TRANSITION not_3621:
NOT MP.ST03.SGM_3621
END_TRANSITION

TRANSITION StateOk:
(*ST08_408_Y54_4.State=STATE_OK*)

ST08_400_Y52_5.State=STATE_OK AND
gTipImp
END_TRANSITION

TRANSITION StateOk:
ST08_408_Y54_4.State =STATE_OK AND
gTipImp
END_TRANSITION

TRANSITION StateOk:
(*ST08_408_Y54_4.State=STATE_OK*)

ST08_400_Y52_5.State=STATE_OK AND
gTipImp
END_TRANSITION

TRANSITION StateOk:
ST08_407_Y51_4.State=STATE_OK AND
gTipImp
END_TRANSITION

TRANSITION TrayKompletOut:
NOT ST08_409_B55_5.BitInToCheck AND
gTipImp
END_TRANSITION

TRANSITION InOutlett:
ST08_409_B55_5.BitInToCheck AND
gTipImp
END_TRANSITION

TRANSITION StateOk:
ST08_407_Y51_4.State=STATE_OK AND
NOT ST00_227_S2.BitInToCheck AND
NOT ST00_230_S1.BitInToCheck AND
gTipImp
END_TRANSITION

TRANSITION StateOk:
ST08_404_Y52_0.State=STATE_OK
END_TRANSITION

TRANSITION not_3621:
NOT MP.ST03.SGM_3621
END_TRANSITION

TRANSITION StateOk:
(*ST08_408_Y54_4.State=STATE_OK*)

ST08_400_Y52_5.State=STATE_OK AND
gTipImp
END_TRANSITION

TRANSITION StateOk:
ST08_408_Y54_4.State=STATE_OK

AND gTipImp
END_TRANSITION

TRANSITION StateOk:
(*ST08_408_Y54_4.State=STATE_OK*)

ST08_400_Y52_5.State=STATE_OK
OR
MP.ST03.SGM_3621
END_TRANSITION

TRANSITION with_Motor:
MP.ST08.StapelMotor
END_TRANSITION

TRANSITION busy:
ST08_180_M1.Busy
END_TRANSITION

TRANSITION Done:
ST08_180_M1.Done
END_TRANSITION

TRANSITION StateOk:
ST08_404_Y53_0.State=STATE_OK
END_TRANSITION

TRANSITION StateOk:
 ST08_404_Y53_2.State=STATE_OK
END_TRANSITION
END_PROGRAM

(* POU System/GeneralFunctions/CallGeneralFunctions, ST *)
PROGRAM CallGeneralFunctions
VAR
	gFB_GETLOCALSYSTEMTIME		:	FB_LocalSystemTime;

	SetLocalTime			: 	NT_SetLocalTime;
	SetTimeStruct			:		TIMESTRUCT;
	SetTimePicEnabled		: 	R_TRIG;

	GetLocalAmsNetId		: 	FB_GetLocalAmsNetId;
	FBWritePersistentData	:	WritePersistentData;

	VisuShutDown:NT_Shutdown;

	TonVisuShutDown : TON;
	ShutDownManual:BOOL;
	ExecuteEverySecondAdFirstCycle: BOOL;
	FBSwitchToConfigMode:TC_Config;
	SwitchToConfigMode: BOOL;

	SavePersistentData: BOOL;
	TDValid								:	R_TRIG;
	PDValid								:	R_TRIG;
	wYear: WORD;
	wMonth: WORD;
	wDay: WORD;
	wHour: WORD;
	wMin: WORD;
	wSec: WORD;

(* Generate Pulses *)
	Pulse1000ms					:	GEN_PULSE;
	Pulse0500ms					:	GEN_PULSE;
	Pulse0100ms					:	GEN_PULSE;
	Pulse0050ms					:	GEN_PULSE;
	Pulse0025ms					:	GEN_PULSE;

	PersDatenCopy					:sPersDaten;

END_VAR
ExecuteEverySecondAdFirstCycle:=SystemTaskInfoArr[SystemInfo.runTimeNo].firstCycle;

GetLocalAmsNetId(
	bExecute:= ExecuteEverySecondAdFirstCycle,
	tTimeout:= t#1s,
	AddrString=> LocalAmsNetIdStr,
	AddrBytes=> LocalAmsNetIdArr);

FBSwitchToConfigMode(
	NETID:= LocalAmsNetIdStr,
	SET:= SwitchToConfigMode ,
	TMOUT:=t#10s );


TDValid(CLK:=gTypeDataValid );

(*Schreibe bei einer Änderung*)
PDValid(CLK:=
	(MEMCMP(ADR(PersDatenCopy), ADR(PersDaten), SIZEOF(PersDatenCopy)) <> 0 ) AND
	ModeSelect.Mode <= MODE_AUTO_RUN);

SavePersistentData:=  TDValid.Q OR PDValid.Q OR visu.SavePersistentData;


FBWritePersistentData(
	NETID:='' ,
	PORT:= 801,
	START:= SavePersistentData,
	TMOUT:=t#2000ms );

visu.SavePersistentData:=FALSE;

(*Impuls Generieren*)
Pulse1000ms(ENQ:=TRUE , PTH:=t#1s, 		PTL:= t#1s, 		Q=>vGlbImpuls_1000ms );
Pulse0500ms(ENQ:=TRUE , PTH:=t#500ms, PTL:= t#500ms, 	Q=>vGlbImpuls_0500ms );
Pulse0100ms(ENQ:=TRUE , PTH:=t#100ms, PTL:= t#100ms, 	Q=>vGlbImpuls_0100ms );
Pulse0050ms(ENQ:=TRUE , PTH:=t#50ms, PTL:= t#50ms, 	Q=>vGlbImpuls_0050ms );
Pulse0025ms(ENQ:=TRUE , PTH:=t#25ms, PTL:= t#25ms, 	Q=>vGlbImpuls_0025ms );


(*		Shutdown Visu on USV - Alarm *)

TonVisuShutDown(IN:= ShutDownManual , PT:= t#2s );

VisuShutDown(
	NETID:= '' ,
	DELAY:=3 ,
	START:= TonVisuShutDown.Q,
	TMOUT:=t#20s );

gFB_GETLOCALSYSTEMTIME(
	sNetID:='' ,
	bEnable:=TRUE ,
	dwCycle:=1 );

gVarStrSystemTime:=SYSTEMTIME_TO_STRING(gFB_GETLOCALSYSTEMTIME.systemTime);
gVarDTSystemtime:=SYSTEMTIME_TO_DT(gFB_GETLOCALSYSTEMTIME.SystemTime);
gVarSystemtime:=gFB_GETLOCALSYSTEMTIME.systemTime;

wYear:=gVarSystemtime.wYear;
wMonth:=gVarSystemtime.wMonth;
wDay:=gVarSystemtime.wDay;
wHour:=gVarSystemtime.wHour;
wMin:=gVarSystemtime.wMinute;
wSec:=gVarSystemtime.wSecond;
gVarStrSystemTime:='';
IF 	wDay<10 THEN
	gVarStrSystemTime:=CONCAT(gVarStrSystemTime ,WORD_TO_STRING(0));
END_IF
gVarStrSystemTime:=CONCAT(gVarStrSystemTime ,WORD_TO_STRING(wDay));
gVarStrSystemTime:=CONCAT(gVarStrSystemTime , '.');
IF 	wMonth<10 THEN
	gVarStrSystemTime:=CONCAT(gVarStrSystemTime ,WORD_TO_STRING(0));
END_IF
gVarStrSystemTime:=CONCAT(gVarStrSystemTime ,WORD_TO_STRING(wMonth));
gVarStrSystemTime:=CONCAT(gVarStrSystemTime , '.');
gVarStrSystemTime:=CONCAT(gVarStrSystemTime ,WORD_TO_STRING(wYear));

gVarStrSystemTime:=CONCAT(gVarStrSystemTime , ' ');
IF 	wHour<10 THEN
	gVarStrSystemTime:=CONCAT(gVarStrSystemTime ,WORD_TO_STRING(0));
END_IF
gVarStrSystemTime:=CONCAT(gVarStrSystemTime ,WORD_TO_STRING(wHour));
gVarStrSystemTime:=CONCAT(gVarStrSystemTime , ':');
IF 	wMin<10 THEN
	gVarStrSystemTime:=CONCAT(gVarStrSystemTime ,WORD_TO_STRING(0));
END_IF
gVarStrSystemTime:=CONCAT(gVarStrSystemTime ,WORD_TO_STRING(wMin));
gVarStrSystemTime:=CONCAT(gVarStrSystemTime , ':');
IF 	wSec<10 THEN
	gVarStrSystemTime:=CONCAT(gVarStrSystemTime ,WORD_TO_STRING(0));
END_IF
gVarStrSystemTime:=CONCAT(gVarStrSystemTime ,WORD_TO_STRING(wSec));

SetTimePicEnabled(CLK:= currentVisu='MP_DATE' );

IF 	SetTimePicEnabled.Q THEN
	SetTimeStruct:=gVarSystemtime;
END_IF

SetLocalTime(
	NETID:= '',
	TIMESTR:= SetTimeStruct,
	TMOUT:= t#10s);
END_PROGRAM

(* POU System/HelpFunctions/GEN_PULSE, ST *)
FUNCTION_BLOCK GEN_PULSE
VAR_INPUT
	ENQ 		: BOOL := TRUE;
	PTH 		:TIME;
	PTL 		:TIME;
END_VAR
VAR_OUTPUT
	Q 			:BOOL;
	Q_FP		:BOOL;
END_VAR
VAR
	ein			:TIME;
	aus			:TIME;
	cyc			:TIME;
	init			:BOOL;
	Q_RTRIG	:R_TRIG;
END_VAR

(*GEN_PULSE uses the internal sps timer to generate a continuous output waveform with programmable high and low time.
the accuracy of gen_pulse is depending on the system timer.
when time is 0 the high and low times are exactly one cycle.
ENQ = TRUE will start and ENQ = FALSE will stop the generator.*)
(* read system timer *)
cyc:=DWORD_TO_TIME(SystemTaskInfoArr[SystemInfo.runTimeNo].cycleTime/10000);
IF 	NOT init THEN
	init:=TRUE;
	aus:=t#0s;
	ein:=t#0s;

END_IF;
IF 	enq AND init THEN
	IF ein<= pth THEN
		ein:=ein+cyc;
		q:=TRUE;
	ELSE
		q:=FALSE;
		aus:=aus+cyc;
		IF 	aus>=ptl THEN
			init:=FALSE;
		END_IF;
	END_IF;

ELSE
	Q := FALSE;
END_IF;

Q_RTRIG(CLK:=Q , Q=>Q_FP );
END_FUNCTION_BLOCK

(* POU zLibrary/ept/Programmbausteine/ST_UPS, ST *)
PROGRAM ST_UPS
VAR_INPUT
	b_Ups				: BOOL;
END_VAR
VAR_IN_OUT

END_VAR
VAR_OUTPUT
END_VAR
VAR
	fb_state_entry		: ST_StateEntry;

	nLastErrID			: UDINT;

	fbGetUpsStatus		: FB_GetUPSStatus;

	bm_ReplaceBattery 	: BOOL;
	bm_NoPower 		: BOOL;
	bm_StatusNotValid 	: BOOL;
	bm_Check			: BOOL;
	fb_rTrig_ReplaceBattery 	: R_TRIG;
	fb_rTrig_NoPower 		: R_TRIG;
	fb_rTrig_StatusNotValid 	: R_TRIG;
	fb_rTrig_Check 			: R_TRIG;
	fb_rTrig_Reset			: R_TRIG;

	bmError				: ErrorStruct;

	FB_ReadXmlLineMsg		:FB_ReadXmlLine;
	tmpErrorText				:STRING;

END_VAR
(*======================================================
   ST: ST_UPS
 ------------------------------------------------------
   Auth: 	Thomas Vilgis    						 
   Date: 	21.06.2018    						     
   Rev.: 		1.0	
   Desc:		Der Baustein liest den Status des Akkupacks aus.
			Die restliche Akkulaufzeit in Minuten kann abgefragt werden.
			Wenn der Akkupack getauscht werden muss wird angezeigt.
			Wenn sich der PC im Netzbetrieb befindet wird angezeigt.
   Historie: 	1.0

 ========================================================*)

fb_state_entry(	i16_pos:= 1);

CASE fb_state_entry.i16_step OF
(*=======================================================*)
	INIT_OBJ:

			fb_state_entry.i16_next_step := INIT;


(*=======================================================*)
	INIT:
		IF fb_state_entry.E THEN

			bm_ReplaceBattery := FALSE;
			bm_NoPower := FALSE;
			bm_StatusNotValid := FALSE;
			bm_Check:= FALSE;
			fbGetUpsStatus.bEnable := FALSE;
		END_IF

		(*-----------------------Weiterschaltbedingungen----------------------------*)
		fb_state_entry.i16_next_step := BEREIT;

(*=======================================================*)
	BEREIT:
		IF 	fb_state_entry.E THEN
			;
		END_IF

		fbGetUpsStatus.bEnable := b_Ups;

		(*-----------------------Weiterschaltbedingungen----------------------------*)
		IF b_Ups THEN
			IF 	fbGetUpsStatus.bValid THEN
				fb_state_entry.i16_next_step := 110;
			ELSIF
				fb_state_entry.fb_ton_Step.ET > t#20s THEN
				bm_StatusNotValid := TRUE;
				fb_state_entry.i16_next_step := FEHLER;
			END_IF
		END_IF

		IF 	fb_state_entry.X THEN
			;
		END_IF

(*=======================================================*)
	110:	(* Evaluation *)

		(*-----------------------Weiterschaltbedingungen----------------------------*)
		IF fbGetUpsStatus.bValid THEN
			IF NOT fbGetUpsStatus.bError THEN
				CASE fbGetUpsStatus.stStatus.eBatteryStatus OF
					BatteryUnknownStatus:	(*Der Akkustatus ist unbekannt*)
						;
					BatteryOk:			(*Der Akku ist in Ordnung*)
						bm_ReplaceBattery := FALSE;
					BatteryReplace:		(*Der Akku sollte gewechselt werden*)
						bm_ReplaceBattery := TRUE;
				END_CASE

				CASE fbGetUpsStatus.stStatus.eCommStatus OF
					UpsCommUnknownStatus:	(*Kommunikationsstatus zur USV-Hardware ist unbekannt*)
						;
					UpsCommOk:		(*Kommunikation zur USV-Hardware ist hergestellt*)
						;
					UpsCommFailed:		(*Kommunikation zur USV wurde unterbrochen*)
						;
				END_CASE

				CASE fbGetUpsStatus.stStatus.ePowerStatus OF
					PowerUnknownStatus:	(*Der Status der Stromversorgung ist unbekannt*)
						;
					PowerOnLine:		(*Das Gerät befindet sich im Netzbetrieb*)
						bm_NoPower := FALSE;
					PowerOnBattery:	(*Stromausfall ist aufgetreten und das Gerät befindet sich im Akkubetrieb*)
						bm_NoPower := TRUE;
				END_CASE
			ELSE
				nLastErrID := fbGetUpsStatus.nErrId;
				fb_state_entry.i16_next_step := FEHLER;
			END_IF
		ELSE
			bm_StatusNotValid := TRUE;
			fb_state_entry.i16_next_step := FEHLER;
		END_IF

(*=======================================================*)
	FEHLER:	 fb_state_entry.s_debugtext:=CONCAT('Error ID: ',UDINT_TO_STRING(nLastErrID));

		IF fb_state_entry.E THEN
			fbGetUpsStatus.bEnable := FALSE;
		END_IF

		(*-----------------------Weiterschaltbedingungen----------------------------*)
		IF 	(fb_state_entry.fb_ton_Step.Q  AND bm_StatusNotValid) OR
			gResetAll THEN
			fb_state_entry.i16_next_step := INIT;
		END_IF

END_CASE

fb_state_entry(i16_pos:= 2 );

fbGetUpsStatus(
	sNetId:= ,	(* wenn in AmsNetId nichts drin steht, wird immer die lokale genommen*)
	nPort:= 0,
	bEnable:= ,
	bValid=> ,
	bError=> ,
	nErrId=> ,
	stStatus=> );

(*Checks zurücksetzen*)
fb_rTrig_Reset(CLK:=gResetAll);
IF fb_rTrig_Reset.Q THEN
	CheckBounds_ErrCnt:=0;
	CheckByteZeroDiv_ErrCnt:=0;
	CheckDWordZeroDiv_ErrCnt:=0;
	CheckRealZeroDiv_ErrCnt:=0;
	CheckWordZeroDiv_ErrCnt:=0;
	CheckRangeSigned_ErrCnt:=0;
	CheckRangeUnsigned_ErrCnt:=0;
END_IF

bm_Check:=ABS(
	CheckBounds_ErrCnt+
	CheckByteZeroDiv_ErrCnt+
	CheckDWordZeroDiv_ErrCnt+
	CheckRealZeroDiv_ErrCnt+
	CheckWordZeroDiv_ErrCnt+
	CheckRangeSigned_ErrCnt+
	CheckRangeUnsigned_ErrCnt	)  > 2 ;

(* Generate information Errorlog *)
fb_rTrig_ReplaceBattery(CLK:=bm_ReplaceBattery);
fb_rTrig_NoPower(CLK:=bm_NoPower);
fb_rTrig_StatusNotValid(CLK:=bm_StatusNotValid);
fb_rTrig_Check(CLK:=bm_Check);

IF 	fb_rTrig_ReplaceBattery.Q THEN
	tmpErrorText:='bm_ReplaceBattery';					(*USV Aku defekt! =>tauschen*)
	bmError.DateTime:= gVarDTSystemtime;
END_IF
IF	fb_rTrig_NoPower.Q THEN
	tmpErrorText:='bm_NoPower';						(*Stromausfall Steuerung wird von der USV versorgt!*)
	bmError.DateTime:= gVarDTSystemtime;
END_IF
IF	fb_rTrig_StatusNotValid.Q THEN
	tmpErrorText:='bm_StatusNotValid';					(*USV Status kann nicht ausgelesen werden*)
	bmError.DateTime:= gVarDTSystemtime;
END_IF
IF	fb_rTrig_Check.Q THEN
	tmpErrorText:='bm_Check';							(*Error Check's*)
	bmError.DateTime:= gVarDTSystemtime;
END_IF

IF 	bm_ReplaceBattery OR
	bm_NoPower OR
	bm_StatusNotValid OR
	bm_Check THEN
	bmError.Typ:= 1;										(* 0=red 1:=orange 2:=blue *)
	bmError.No:= 1;
	ErrorHandler.AddError(ErrorToAdd:=bmError,sVisu:=Visu.ErrorHandler);
END_IF

FB_ReadXmlLineMsg(
	Prefix:= 'MSG',
	ID:= tmpErrorText,
	File:= 'MSG.xml',
	Text=>bmError.Text);
END_PROGRAM

(* POU zLibrary/ept/Programmbausteine/ST_CPU, ST *)
PROGRAM ST_CPU
VAR_INPUT
	iNumberOfFan			: INT := 1;
	iNumberOfCPU			: INT := 1;
	iLANIdx					: USINT;
END_VAR
VAR_IN_OUT

END_VAR
VAR_OUTPUT
	st_ctrl_out				: struct_ctrl_out;
	LNG					: enum_Lng:=DE;
END_VAR
VAR
	fb_ton_quitt				: TON;
	fb_state_entry			: ST_StateEntry;

	fbGetCPUUsage			: FB_MDP_CPU_Read;

	fbMDPNICRead			: FB_MDP_NIC_Read;	(* IP and MAC address *)

	fbGetRealTimeUsage	: TC_CpuUsage;

	fbGetHostName			:FB_GetHostName;

	nLastErrID	:UDINT;

	(* request cpu temperature *)
	fbGetCpuTemp			:FB_MDP_ReadElement;
	stMDP_Addr			:ST_MDP_Addr;		(* includes all address parameters without the Dynamic Module Id *)

	iCpu					:USINT;

	fbGetMainboardInfo		:FB_MDP_ReadElement;
	(* request fan speed *)
	fbGetFanSpeed			:FB_MDP_ReadElement;

	iFan					:USINT;

	fbGetTcInfo				:FB_MDP_TwinCAT_Read;

	b_temp								: BOOL;
	bm_CpuTemperatureToHigh 			: BOOL;
	bm_CpuUsageToHigh 				: BOOL;
	bm_FanSpeedToLow 				: BOOL;
	bm_RealTimeUsageToHigh 			: BOOL;
	bm_MainboardTemperatureToHigh 	: BOOL;

	(* visu *)
	s_Lng_Ip				: sData_Str:=(Description:='s_Lng_Ip');
	s_actual_IP_Adress		: sData_Str:=(Description:='s_actual_IP_Adress');
	b_DHCP				: sData_b:=(Description:='b_DHCP');
	s_Host_Name			: sData_Str:=(Description:='s_Host_Name');
	s_MAC_Address			: sData_Str:=(Description:='s_MAC_Address');
	s_Subnet_Mask			: sData_Str:=(Description:='s_Subnet_Mask');
	s_AMSNetId			: sData_Str:=(Description:='s_AMSNetId');
	i_Build					: sData_i16:=(Description:='i_Build', Unit:='no');
	i_RealTimeUsage		: sData_i16:=(Description:='i_RealTimeUsage', Unit:='%');
	i_FanSpeed				: ARRAY [0..4] OF sData_i16:=
										(Description:='i_FanSpeed[0]', Unit:='U/min'),
										(Description:='i_FanSpeed[1]', Unit:='U/min'),
										(Description:='i_FanSpeed[2]', Unit:='U/min'),
										(Description:='i_FanSpeed[3]', Unit:='U/min');
	i_CpuTemperature		: ARRAY [0..4] OF sData_i16:=
										(Description:='i_CpuTemperature[0]', Unit:='°C'),
										(Description:='i_CpuTemperature[1]', Unit:='°C'),
										(Description:='i_CpuTemperature[2]', Unit:='°C'),
										(Description:='i_CpuTemperature[3]', Unit:='°C');
	i_CpuUsage			: ARRAY [0..4] OF sData_i16:=
										(Description:='i_CpuUsage[0]', Unit:='%'),
										(Description:='i_CpuUsage[1]', Unit:='%'),
										(Description:='i_CpuUsage[2]', Unit:='%'),
										(Description:='i_CpuUsage[3]', Unit:='%');
	i_MainboardTemperature	: sData_i16:=(Description:='i_MainboardTemperature', Unit:='°C');


END_VAR
VAR_TEMP
	i				:INT;
END_VAR
(*======================================================
   ST: ST_CPU
 ------------------------------------------------------
   Auth: 	Thomas Vilgis    						 
   Date: 	24.05.2018    						     
   Rev.: 		1.0	
   Desc:		Der Baustein liest am Anfang den Hostnamen, die MAC-Adresse, IP-Adresse
			und die TwinCAT Infos aus. Danach werden in einem bestimmten Intervall
			die Echtzeitauslastung des TwinCATs, die CPU-Auslastung und die 
			CPU-Temperaturen ausgelesen. Außerdem die Drehzahl der Lüfter.

   Historie: 	
   Auth: 	Werner Friedl    						 
   Date: 	01.03.2021
		LNG auslesen aus der IP 
		16,17 und 18 => DE
		19 und 20 => CZ
		22 => EN
 ========================================================*)
(* Zeiten *)
fb_ton_quitt(IN:= , PT:= t#100ms, Q=> , ET=> );

(* Flanken *)

(* ======================================Schrittkette======================================== *)
fb_state_entry(	i16_pos:= 1);

CASE fb_state_entry.i16_step OF
(*=======================================================*)
	INIT_OBJ:
		IF	TD.ArtNo <> '' AND
			CURRENTLANGUAGE <> '' THEN
			IF	CURRENTLANGUAGE = 'DE' THEN
				s_Lng_Ip.str:='DE';
				LNG:=DE;
			ELSIF
				CURRENTLANGUAGE = 'EN' THEN
				s_Lng_Ip.str:='EN';
				LNG:=EN;
			ELSIF
				CURRENTLANGUAGE = 'CZ' THEN
				s_Lng_Ip.str:='CZ';
				LNG:=CZ;
			END_IF
			fb_state_entry.i16_next_step := INIT;
		END_IF

(*=======================================================*)
	INIT:
		IF fb_state_entry.E THEN
			fb_ton_quitt.IN := FALSE;
			st_ctrl_out.b_fehler := FALSE;
			st_ctrl_out.b_bereit := FALSE;
			st_ctrl_out.b_fertig := FALSE;
			st_ctrl_out.b_busy := FALSE;

			bm_CpuTemperatureToHigh := FALSE;
			bm_CpuUsageToHigh := FALSE;
			bm_FanSpeedToLow := FALSE;
			bm_RealTimeUsageToHigh := FALSE;
			bm_MainboardTemperatureToHigh := FALSE;

			fbGetCPUUsage.bExecute := FALSE;
			fbGetRealTimeUsage.START := FALSE;
			fbMDPNICRead.bExecute := FALSE;
			fbGetHostName.bExecute := FALSE;
			fbGetCpuTemp.bExecute := FALSE;
			fbGetFanSpeed.bExecute := FALSE;
			fbGetTcInfo.bExecute := FALSE;
			fbGetMainboardInfo.bExecute := FALSE;
			nLastErrID:=0;
			iLANIdx:=INT_TO_USINT(MP.ST00.LAN_no.i16);			(*0=LAN1, 1=LAN2, 2=LAN-USB*)
		END_IF

		(*-----------------------Weiterschaltbedingungen----------------------------*)
		IF 	fb_state_entry.fb_ton_Step.ET > t#10s THEN
			fb_state_entry.i16_next_step := 20;
		END_IF

(*=======================================================*)
	20:	fb_state_entry.s_debugtext:='Get Host Name ';

		IF fb_state_entry.E THEN
			fbGetHostName.bExecute := TRUE;
		END_IF

		(*-----------------------Weiterschaltbedingungen----------------------------*)
		IF fbGetHostName.bBusy THEN
			fbGetHostName.bExecute := FALSE;
			fb_state_entry.i16_next_step := 30;
		END_IF

(*=======================================================*)
	30:	fb_state_entry.s_debugtext:='Get Host Name  ';

		(*-----------------------Weiterschaltbedingungen----------------------------*)
		IF NOT fbGetHostName.bBusy THEN
			IF NOT fbGetHostName.bError THEN
				fb_state_entry.i16_next_step := 40;
			ELSE
				nLastErrID := fbGetHostName.nErrID;
				fb_state_entry.i16_next_step := FEHLER;
			END_IF
		END_IF

(*=======================================================*)
	40:	fb_state_entry.s_debugtext:='Get IP Adress und MAC-Adress';

		IF fb_state_entry.E THEN
			fbMDPNICRead.bExecute := TRUE;
		END_IF

		(*-----------------------Weiterschaltbedingungen----------------------------*)
		IF fbMDPNICRead.bBusy THEN
			fbMDPNICRead.bExecute := FALSE;
			fb_state_entry.i16_next_step := 50;
		END_IF

(*=======================================================*)
	50:	fb_state_entry.s_debugtext:='Get IP Adress und MAC-Adress ';

		(*-----------------------Weiterschaltbedingungen----------------------------*)
		IF 	NOT fbMDPNICRead.bBusy THEN
			IF NOT fbMDPNICRead.bError THEN
				fb_state_entry.i16_next_step := 60;
			ELSE
				nLastErrID := fbMDPNICRead.nErrID;
				fb_state_entry.i16_next_step := FEHLER;
			END_IF
		END_IF

(*=======================================================*)
	60:	fb_state_entry.s_debugtext:='Get IP Adress und MAC-Adress ';

		(*-----------------------Weiterschaltbedingungen----------------------------*)
		IF fb_state_entry.E THEN
			s_actual_IP_Adress.str := fbMDPNICRead.stMDP_ModuleContent.sIPAddress;
			s_MAC_Address.str := fbMDPNICRead.stMDP_ModuleContent.sMACAddress;
			s_Subnet_Mask.str := fbMDPNICRead.stMDP_ModuleContent.sSubnetMask;
			b_DHCP.b := fbMDPNICRead.stMDP_ModuleContent.bDHCP;
			s_Lng_Ip.str:=s_actual_IP_Adress.str;
			s_Lng_Ip.str:=RIGHT(	s_Lng_Ip.str,	LEN(s_Lng_Ip.str) - FIND(s_Lng_Ip.str,'.')	);
			s_Lng_Ip.str:=LEFT(s_Lng_Ip.str, 2);
			fb_state_entry.i16_next_step := 70;
			IF	s_Lng_Ip.str = '16' OR s_Lng_Ip.str = '17' OR s_Lng_Ip.str = '18' THEN	(*Peiting, Buching, Augsburg*)
				s_Lng_Ip.str:=CONCAT(s_Lng_Ip.str,' => DE');
				LNG:= DE;
				MP.ST00.LAN_no.i16:=USINT_TO_INT(iLANIdx);			(*0=LAN1, 1=LAN2, 2=LAN-USB*)
			ELSIF
				s_Lng_Ip.str = '22' THEN
				s_Lng_Ip.str:=CONCAT(s_Lng_Ip.str,' => EN');
				LNG:= EN;
				MP.ST00.LAN_no.i16:=USINT_TO_INT(iLANIdx);			(*0=LAN1, 1=LAN2, 2=LAN-USB*)
			ELSIF
				s_Lng_Ip.str = '19' OR s_Lng_Ip.str = '20' THEN
				s_Lng_Ip.str:=CONCAT(s_Lng_Ip.str,' => CZ');
				LNG:= CZ;
				MP.ST00.LAN_no.i16:=USINT_TO_INT(iLANIdx);			(*0=LAN1, 1=LAN2, 2=LAN-USB*)
			ELSE
				IF	iLANIdx<2 THEN
						iLANIdx:=iLANIdx + 1;
						fb_state_entry.i16_next_step := 40;
				END_IF
			END_IF
	END_IF

(*=======================================================*)
	70:	fb_state_entry.s_debugtext:='Get TwinCAT Info ';
		IF fb_state_entry.E THEN
			fbGetTcInfo.bExecute := TRUE;
		END_IF

		(*-----------------------Weiterschaltbedingungen----------------------------*)
		IF fbGetTcInfo.bBusy THEN
			fbGetTcInfo.bExecute := FALSE;
			fb_state_entry.i16_next_step := 80;
		END_IF

(*=======================================================*)
	80:	fb_state_entry.s_debugtext:='Get TwinCAT Info ';

		(*-----------------------Weiterschaltbedingungen----------------------------*)
		IF NOT fbGetTcInfo.bBusy THEN
			IF NOT fbGetTcInfo.bError THEN
				s_AMSNetId.str := fbGetTcInfo.stMDP_ModuleContent.sAmsNETid;
				i_Build.i16 := fbGetTcInfo.stMDP_ModuleContent.iBuild;
				fb_state_entry.i16_next_step := BEREIT;
			ELSE
				nLastErrID := fbGetTcInfo.nErrID;
				fb_state_entry.i16_next_step := FEHLER;
			END_IF
		END_IF

(*=======================================================*)
	BEREIT:	fb_state_entry.s_debugtext:='warte auf Start';

		IF fb_state_entry.E THEN
			st_ctrl_out.b_bereit := TRUE;
		END_IF

		(*-----------------------Weiterschaltbedingungen----------------------------*)
		IF 	iLANIdx <> INT_TO_USINT(MP.ST00.LAN_no.i16) THEN
			fb_state_entry.i16_next_step := INIT;
		END_IF

		IF 	fb_state_entry.fb_ton_Step.ET > t#10s THEN
			iCpu := 1;
			iFan := 1;
			fb_state_entry.i16_next_step := 110;
		END_IF

		IF fb_state_entry.X THEN
			st_ctrl_out.b_bereit := FALSE;
			st_ctrl_out.b_fertig := FALSE;
			st_ctrl_out.b_busy := TRUE;
		END_IF

(*=======================================================*)
	110:	fb_state_entry.s_debugtext:='Get Real Time Usage';

		IF fb_state_entry.E THEN
			fbGetRealTimeUsage.START := TRUE;
		END_IF

		(*-----------------------Weiterschaltbedingungen----------------------------*)
		IF 	fbGetRealTimeUsage.BUSY THEN
			fbGetRealTimeUsage.START := FALSE;
			fb_state_entry.i16_next_step := 120;
		END_IF

(*=======================================================*)
	120:	fb_state_entry.s_debugtext:='Get Real Time Usage';

		(*-----------------------Weiterschaltbedingungen----------------------------*)
		IF NOT fbGetRealTimeUsage.BUSY THEN
			IF NOT fbGetRealTimeUsage.ERR THEN
				i_RealTimeUsage.i16 := UDINT_TO_INT(fbGetRealTimeUsage.USAGE);
				fb_state_entry.i16_next_step := 130;
			ELSE
				nLastErrID := fbGetRealTimeUsage.ERRID;
				fb_state_entry.i16_next_step := FEHLER;
			END_IF
		END_IF

(*=======================================================*)
	130:	fb_state_entry.s_debugtext:='Get CPU Usage ';

		IF fb_state_entry.E THEN
			fbGetCPUUsage.bExecute := TRUE;
			fbGetCPUUsage.iModIdx := iCpu-1;		(* number of cpu *)
		END_IF

		(*-----------------------Weiterschaltbedingungen----------------------------*)
		IF fbGetCPUUsage.bBusy THEN
			fbGetCPUUsage.bExecute := FALSE;
			fb_state_entry.i16_next_step := 140;
		END_IF

(*=======================================================*)
	140:	fb_state_entry.s_debugtext:='Get CPU Usage';

		(*-----------------------Weiterschaltbedingungen----------------------------*)
		IF NOT fbGetCPUUsage.bBusy THEN
			IF NOT fbGetCPUUsage.bError THEN
				i_CpuUsage[iCpu-1].i16 := fbGetCPUUsage.stMDP_ModuleContent.iCPUusage;
				fb_state_entry.i16_next_step := 150;
			ELSE
				nLastErrID := fbGetCPUUsage.nErrId;
				fb_state_entry.i16_next_step := FEHLER;
			END_IF
		END_IF

(*=======================================================*)
	150:	fb_state_entry.s_debugtext:='Get CPU temperature';

		IF fb_state_entry.E THEN
			stMDP_Addr.nArea := INT_TO_BYTE(eMDP_Area_ConfigArea);
			stMDP_Addr.nTableId := 1;
			stMDP_Addr.nSubIdx := 3;			(* SubIndex 3 = cpu temperature *)
			fbGetCpuTemp.iModIdx := iCpu-1;		(* number of cpu *)
			fbGetCpuTemp.pDstBuf := ADR(i_CpuTemperature[iCpu-1].i16);
			fbGetCpuTemp.cbDstBufLen := SIZEOF(i_CpuTemperature[iCpu-1].i16);
			fbGetCpuTemp.bExecute := TRUE;
		END_IF

		(*-----------------------Weiterschaltbedingungen----------------------------*)
		IF fbGetCpuTemp.bBusy THEN
			fbGetCpuTemp.bExecute := FALSE;
			fb_state_entry.i16_next_step := 160;
		END_IF

(*=======================================================*)
	160:	fb_state_entry.s_debugtext:='Get CPU temperature';

		(*-----------------------Weiterschaltbedingungen----------------------------*)
		IF NOT fbGetCpuTemp.bBusy THEN
			IF NOT fbGetCpuTemp.bError THEN
				fb_state_entry.i16_next_step := 170;
			ELSE
				nLastErrID := fbGetCpuTemp.nErrId;
				fb_state_entry.i16_next_step := FEHLER;
			END_IF
		END_IF

(*=======================================================*)
	170:	fb_state_entry.s_debugtext:='warte';	(* Count CPU  *)
		IF fb_state_entry.E THEN
			iCpu := iCpu + 1;
		END_IF

		(*-----------------------Weiterschaltbedingungen----------------------------*)
		IF iCpu > iNumberOfCPU THEN
			fb_state_entry.i16_next_step := 180;
		ELSE
			fb_state_entry.i16_next_step := 130;
		END_IF

(*=======================================================*)
	180:	fb_state_entry.s_debugtext:='Get Fan speed ';

		IF fb_state_entry.E THEN
			stMDP_Addr.nArea := INT_TO_BYTE(eMDP_Area_ConfigArea);
			stMDP_Addr.nTableId := 1;
			stMDP_Addr.nSubIdx := 1;			(* SubIndex 1 = fan speed *)
			fbGetFanSpeed.iModIdx := iFan-1;		(* number of fan *)
			fbGetFanSpeed.pDstBuf := ADR(i_FanSpeed[iFan-1].i16);
			fbGetFanSpeed.cbDstBufLen := SIZEOF(i_FanSpeed[iFan-1].i16);
			fbGetFanSpeed.bExecute := TRUE;
		END_IF

		(*-----------------------Weiterschaltbedingungen----------------------------*)
		IF fbGetFanSpeed.bBusy THEN
			fbGetFanSpeed.bExecute := FALSE;
			fb_state_entry.i16_next_step := 190;
		END_IF

(*=======================================================*)
	190:	fb_state_entry.s_debugtext:='Get Fan speed';

		(*-----------------------Weiterschaltbedingungen----------------------------*)
		IF NOT fbGetFanSpeed.bBusy THEN
			IF NOT fbGetFanSpeed.bError THEN
				fb_state_entry.i16_next_step := 200;
			ELSE
				nLastErrID := fbGetFanSpeed.nErrId;
				fb_state_entry.i16_next_step := FEHLER;
			END_IF
		END_IF

(*=======================================================*)
	200:	fb_state_entry.s_debugtext:='Count Fan';

		IF fb_state_entry.E THEN
			iFan := iFan + 1;
		END_IF

		(*-----------------------Weiterschaltbedingungen----------------------------*)
		IF iFan > iNumberOfFan THEN
			fb_state_entry.i16_next_step := 210;
		ELSE
			fb_state_entry.i16_next_step := 180;
		END_IF

(*=======================================================*)
	210:	fb_state_entry.s_debugtext:='Get Mainboard Temperature';

		IF fb_state_entry.E THEN
			stMDP_Addr.nArea := INT_TO_BYTE(eMDP_Area_ConfigArea);
			stMDP_Addr.nTableId := 1;
			stMDP_Addr.nSubIdx := 10;			(* SubIndex 1 = mainboard temperature *)
			fbGetMainboardInfo.pDstBuf := ADR(i_MainboardTemperature.i16);
			fbGetMainboardInfo.cbDstBufLen := SIZEOF(i_MainboardTemperature.i16);
			fbGetMainboardInfo.bExecute := TRUE;
		END_IF

		(*-----------------------Weiterschaltbedingungen----------------------------*)
		IF fbGetMainboardInfo.bBusy THEN
			fbGetMainboardInfo.bExecute := FALSE;
			fb_state_entry.i16_next_step := 220;
		END_IF

(*=======================================================*)
	220:	fb_state_entry.s_debugtext:='GetMainboard Temperature ';

		(*-----------------------Weiterschaltbedingungen----------------------------*)
		IF NOT fbGetMainboardInfo.bBusy THEN
			IF NOT fbGetMainboardInfo.bError THEN
				fb_state_entry.i16_next_step := 230;
			ELSE
				nLastErrID := fbGetMainboardInfo.nErrId;
				fb_state_entry.i16_next_step := FEHLER;
			END_IF
		END_IF

(*=======================================================*)
	230:	fb_state_entry.s_debugtext:='evaluation';

		IF fb_state_entry.E THEN
			b_temp := FALSE;
			FOR i:=0 TO iNumberOfFan-1 DO
				IF i_FanSpeed[i].i16 < 5500 THEN
					b_temp := TRUE;
				END_IF
			END_FOR
			bm_FanSpeedToLow := b_temp;

			b_temp := FALSE;
			FOR i:=0 TO iNumberOfCPU-1 DO
				IF i_CpuTemperature[i].i16 > 80 THEN
					b_temp := TRUE;
				END_IF
			END_FOR
			bm_CpuTemperatureToHigh := b_temp;

			b_temp := FALSE;
			FOR i:=0 TO iNumberOfCPU-1 DO
				IF i_CpuUsage[i].i16 > 70 THEN
					b_temp := TRUE;
				END_IF
			END_FOR
			bm_CpuUsageToHigh := b_temp;

			bm_RealTimeUsageToHigh := i_RealTimeUsage.i16 > 30;

			bm_MainboardTemperatureToHigh := i_MainboardTemperature.i16 > 70;
		END_IF

		(*-----------------------Weiterschaltbedingungen----------------------------*)
		st_ctrl_out.b_fertig := TRUE;
		st_ctrl_out.b_busy := FALSE;
		fb_state_entry.i16_next_step := BEREIT;

(*=======================================================*)
	STOP, FEHLER:fb_state_entry.s_debugtext:=CONCAT('Error ID: ',UDINT_TO_STRING(nLastErrID));

		IF fb_state_entry.E THEN
			st_ctrl_out.b_fehler := fb_state_entry.i16_next_step = FEHLER;
			st_ctrl_out.b_gestoppt := fb_state_entry.i16_next_step = STOP;
			fb_ton_quitt.IN := FALSE;

		END_IF

		(*-----------------------Weiterschaltbedingungen----------------------------*)
		IF 	fb_state_entry.fb_ton_Step.ET > t#2s THEN
			st_ctrl_out.b_fehler := FALSE;
			st_ctrl_out.b_gestoppt := FALSE;
			fb_ton_quitt.IN := TRUE;
		END_IF
	
		IF 	fb_ton_quitt.Q THEN
			fb_ton_quitt.IN := FALSE;
			fb_state_entry.i16_next_step := INIT;
		END_IF

END_CASE

fb_state_entry(i16_pos:= 2 );

fbGetFanSpeed(
	bExecute:= ,
	stMDP_Addr:= stMDP_Addr,
	eModuleType:= eMDP_ModT_Fan,
	iModIdx:= ,
	tTimeout:= ,	(* default 5s *)
	sAmsNetId:= , (* wenn in AmsNetId nichts drin steht, wird immer die lokale genommen*)
	bBusy=> ,
	bError=> ,
	nErrID=> ,
	nCount=> ,
	stMDP_DynAddr=> ,
	iModuleTypeCount=> ,
	iModuleCount=> );

fbGetCpuTemp(
	bExecute:= ,
	stMDP_Addr:= stMDP_Addr,
	eModuleType:= eMDP_ModT_CPU,
	iModIdx:= ,
	pDstBuf     := ,
	cbDstBufLen := ,
	tTimeout:= ,	(* default 5s *)
	sAmsNetId:= , (* wenn in AmsNetId nichts drin steht, wird immer die lokale genommen*)
	bBusy=> ,
	bError=> , 
	nErrID=> ,
	nCount=> ,
	stMDP_DynAddr=> ,
	iModuleTypeCount=> ,
	iModuleCount=> );

fbGetCPUUsage(
	bExecute:= ,
	tTimeout:= ,	(* default 5s *)
	iModIdx:= ,
	sAmsNetId:= , (* wenn in AmsNetId nichts drin steht, wird immer die lokale genommen*)
	bBusy=> ,
	bError=> ,
	nErrID=> ,
	iErrPos=> ,
	stMDP_ModuleHeader=> ,
	stMDP_ModuleContent=> );

fbMDPNICRead(
	bExecute:= ,
	tTimeout:= , 	(* default 5s *)
	iModIdx:= iLANIdx, 	(*0=EtherCAT, 1=LAN muss aber nicht immer so sein*)
	sAmsNetId:= , (* wenn in AmsNetId nichts drin steht, wird immer die lokale genommen*)
	bBusy=> ,
	bError=> ,
	nErrID=> ,
	iErrPos=> ,
	stMDP_ModuleHeader=> ,
	stMDP_ModuleContent=> );

fbGetRealTimeUsage(
	NETID:= ,(* wenn in AmsNetId nichts drin steht, wird immer die lokale genommen*)
	START:= ,
	TMOUT:= ,	(* default 5s *)
	BUSY=> ,
	ERR=> ,
	ERRID=> ,
	USAGE=> );

fbGetHostName(
	sNetID:= ,(* wenn in AmsNetId nichts drin steht, wird immer die lokale genommen*)
	bExecute:= ,
	tTimeout:= , 	(* default 5s *)
	bBusy=> ,
	bError=> ,
	nErrID=> ,
	sHostName=> s_Host_Name.str);

fbGetTcInfo(
	bExecute:= , 
	tTimeout:= , 	(* default 5s *)
	iModIdx:= , 
	sAmsNetId:= , (* wenn in AmsNetId nichts drin steht, wird immer die lokale genommen*)
	bBusy=> ,
	bError=> , 
	nErrID=> ,
	iErrPos=> ,
	stMDP_ModuleHeader=> , 
	stMDP_ModuleContent=> );

fbGetMainboardInfo(
	bExecute:= ,
	stMDP_Addr:= stMDP_Addr,
	eModuleType:= eMDP_ModT_Mainboard,
	iModIdx:= ,
	pDstBuf:= ,
	cbDstBufLen:= ,
	tTimeout:= , 
	sAmsNetId:= ,(* wenn in AmsNetId nichts drin steht, wird immer die lokale genommen*)
	bBusy=> , 
	bError=> ,
	nErrID=> ,
	nCount=> , 
	stMDP_DynAddr=> , 
	iModuleTypeCount=> ,
	iModuleCount=> );

(*
IF	TD.ArtNo <> '' THEN
	(* Fehlermeldungen und Betriebsmeldungen ab dem Startindex in die globalen Meldungsarrays schreiben *)
	garr_stoermeldungen[st_config.i16_meld_startindex + 0] := FALSE;
	garr_stoermeldungen[st_config.i16_meld_startindex + 1] := FALSE;
	garr_stoermeldungen[st_config.i16_meld_startindex + 2] := FALSE;
	garr_stoermeldungen[st_config.i16_meld_startindex + 3] := FALSE;
	garr_stoermeldungen[st_config.i16_meld_startindex + 4] := FALSE;

	garr_betriebsmeldungen[st_config.i16_meld_startindex + 0] := bm_RealTimeUsageToHigh;
	garr_betriebsmeldungen[st_config.i16_meld_startindex + 1] := bm_CpuTemperatureToHigh;
	garr_betriebsmeldungen[st_config.i16_meld_startindex + 2] := bm_CpuUsageToHigh;
	garr_betriebsmeldungen[st_config.i16_meld_startindex + 3] := bm_FanSpeedToLow;
	garr_betriebsmeldungen[st_config.i16_meld_startindex + 4] := bm_MainboardTemperatureToHigh;

END_IF*)
END_PROGRAM

(* POU zLibrary/ept/ST_AutoCheckIn, ST *)
PROGRAM ST_AutoCheckIn
VAR_INPUT
	i_IntervalDay				: INT;		(*all  X Tagen, 0 = jeden Tag*)
END_VAR
VAR_OUTPUT
END_VAR
VAR
	fb_state_entry			: ST_StateEntry;
	NT_StartProcess 		: NT_StartProcess;
	s_uhrzeit				: STRING;
	s_tmpUhrzeit			: STRING;
	i_DayOfYear			: DINT;
	i_ErrId					: UDINT;
END_VAR
VAR_TEMP
	i						:INT:=1;
END_VAR
VAR CONSTANT
	NO_OF_AUTOCHECKIN	: INT :=5;

 	s_AutoCheckIn			:  ARRAY[1..NO_OF_AUTOCHECKIN] OF STRING:=
											'AutoCheckInDaten.bat',
											'AutoCheckInEpson.bat',
											'',
											'',
											''			;
END_VAR
(*======================================================
   FB: Start AutoCheckIn
 ------------------------------------------------------
   Auth: 		Werner Friedl   						 
   Date: 		10.11.2020  						     
   Rev.: 		1.0	
   Desc:		Mit diesem Programm können Komponenten im Versdog automatisch eingecheckt werden.
			Für den Check in benötigt man einen Bat- Datei. Diese liegt im Projektverzeichnis "Tools" und 
			muss für jede Komponente erstellt werden.
			Wenn mehrere Komponeten Eingecheckt werden sollen muss im Array "s_AutoCheckIn" die
			Bat Datei eingetragen werden.

			- die Input Variable "i_IntervalDay" legt den Seicherintervall in x Tagen fest.
			Wenn das Speichern nicht klappt, dann wird einen Tag später der nächste Versuch gemacht.

		Beispiel Aufruf:
		ST_AutoCheckIn( i_IntervalDay:=7 );

   Historie:   1.0

=======================================================*)

(* Uhrzei *)
s_uhrzeit:='';
s_uhrzeit:=CONCAT(s_uhrzeit, WORD_TO_STRING(gVarSystemtime.wHour));
s_uhrzeit:=CONCAT(s_uhrzeit, ':');
s_uhrzeit:=CONCAT(s_uhrzeit, WORD_TO_STRING(gVarSystemtime.wMinute));
s_uhrzeit:=CONCAT(s_uhrzeit, ':');
s_uhrzeit:=CONCAT(s_uhrzeit, WORD_TO_STRING(gVarSystemtime.wSecond));

(* Tag im Jahr *)
i_DayOfYear:=F_GetDOYOfYearMonthDay( gVarSystemtime.wYear, gVarSystemtime.wMonth, gVarSystemtime.wDay );

fb_state_entry(i16_pos:= 1);

CASE fb_state_entry.i16_step OF

(*=======================================================*)
INIT_OBJ:

	(*-----------------------Weiterschaltbedingungen----------------------------*)
	IF	i_DayOfYear <>0  AND
		fb_state_entry.fb_ton_Step.ET > t#5s THEN
		fb_state_entry.i16_next_step := 5;
	END_IF

(*=======================================================*)
5:
	(*-----------------------Weiterschaltbedingungen----------------------------*)
	IF	TD.ArtNo <>'' AND
		s_uhrzeit <> '00:00:00' AND s_uhrzeit <> ''  THEN
		IF	PersDaten.i_DayOfYearAutoCheckIn > i_DayOfYear THEN
			PersDaten.i_DayOfYearAutoCheckIn:= i_DayOfYear;
		END_IF
			fb_state_entry.i16_next_step := 6;
	END_IF

(*=======================================================*)
6:
	IF fb_state_entry.E THEN
		s_tmpUhrzeit:=s_uhrzeit;
		(*s_tmpUhrzeit:=REPLACE (s_tmpUhrzeit,'00',2,1);*)	(*nur in der Nacht sichern*)
	END_IF

	(*-----------------------Weiterschaltbedingungen----------------------------*)
	IF 	fb_state_entry.fb_ton_Step.ET > t#59s THEN
		IF	PersDaten.i_DayOfYearAutoCheckIn + i_IntervalDay < i_DayOfYear  THEN
			fb_state_entry.i16_next_step:=110;		(*gleich sicher, da das letzte Sichern zu lange her ist*)
		ELSE
			fb_state_entry.i16_next_step:=INIT;
		END_IF
	END_IF

(*=======================================================*)
INIT:
	IF 	fb_state_entry.E THEN
		;
	END_IF

	(*-----------------------Weiterschaltbedingungen----------------------------*)
	fb_state_entry.i16_next_step := BEREIT;

(*=======================================================*)
BEREIT: fb_state_entry.s_debugtext:='warte auf Start';

	IF 	fb_state_entry.E THEN
		;
	END_IF

	(*-----------------------Weiterschaltbedingungen----------------------------*)
	IF 	s_tmpUhrzeit=s_uhrzeit AND
		(PersDaten.i_DayOfYearAutoCheckIn + i_IntervalDay) <= i_DayOfYear THEN
		fb_state_entry.i16_next_step:=110;
	END_IF

	IF 	fb_state_entry.X THEN
		i:=0;
	END_IF

(*=======================================================*)
110:  fb_state_entry.s_debugtext:='Start Autocheckin';

	IF 	fb_state_entry.E THEN
		i:=i+1;
	END_IF

	IF	i = NO_OF_AUTOCHECKIN + 1 OR
		s_AutoCheckIn[i] = '' THEN
		fb_state_entry.i16_next_step:=200;
	ELSE
		fb_state_entry.i16_next_step:=120;
	END_IF

(*=======================================================*)
120:  fb_state_entry.s_debugtext:='Start Autocheckin';

	IF fb_state_entry.E THEN
		NT_StartProcess.START:=TRUE;
	END_IF

	(*-----------------------Weiterschaltbedingungen----------------------------*)
	IF 	NT_StartProcess.BUSY THEN
		fb_state_entry.i16_next_step:=130;
	END_IF

	IF 	fb_state_entry.X THEN
		NT_StartProcess.START:=FALSE;
	END_IF

(*=======================================================*)
130:  fb_state_entry.s_debugtext:='Warte auf fertig Autocheckin';

	IF 	NT_StartProcess.ERR THEN
		i_ErrId:=NT_StartProcess.ERRID;
		fb_state_entry.i16_next_step:=FEHLER;
	ELSIF
	 	fb_state_entry.fb_ton_Step.ET > t#5s AND
		NOT NT_StartProcess.BUSY AND
		NOT NT_StartProcess.ERR THEN
		fb_state_entry.i16_next_step:=110;
	END_IF

(*=======================================================*)
(*=======================================================*)
200:  fb_state_entry.s_debugtext:='Ende';

	(*-----------------------Weiterschaltbedingungen----------------------------*)
	PersDaten.i_DayOfYearAutoCheckIn:=i_DayOfYear;
	fb_state_entry.i16_next_step:=BEREIT;

(*=======================================================*)
STOP, FEHLER:
	IF 	fb_state_entry.E THEN
		IF	i_ErrId <> 0 THEN
		 	fb_state_entry.s_debugtext:=CONCAT('nErrId = ', UDINT_TO_STRING(i_ErrId)	);
		END_IF
		i_ErrId:=0;
	END_IF

	(*-----------------------Weiterschaltbedingungen----------------------------*)
	IF	fb_state_entry.fb_ton_Step.ET>t#1ms THEN
		fb_state_entry.i16_next_step := INIT;
	END_IF

END_CASE

fb_state_entry(i16_pos:= 2 );


(*Aufrufe======================================================*)
NT_StartProcess(
	NETID:='',
	PATHSTR		:='C:\Windows\System32\cmd.exe',
	DIRNAME		:=s_tools_path,
	COMNDLINE	:=CONCAT('/C start /b ', s_AutoCheckIn[i])	,
	START			:=,
	TMOUT			:=DEFAULT_ADS_TIMEOUT);
END_PROGRAM

(* POU zLibrary/ept/MainMenue/ST_MainMenue, ST *)
PROGRAM ST_MainMenue
VAR
	b_init					:BOOL:=FALSE;
	NT_StartProcess 		:NT_StartProcess;

	str_CurrentVisu_TD		:STRING:='TD_01_EDIT';

	FB_BtnTree				:FB_Btn;
END_VAR
IF NOT b_init THEN
	b_init:=TRUE;
END_IF

MainMenue_Btn_Init();
END_PROGRAM
ACTION MainMenue_Btn_Init:
(*=====================================================================*)
FB_BtnTree( Zoom:='MAIN',
			deaktivieren:=FALSE,
			unsichtbar:=FALSE,
			Btn=> Visu.MainMenue.BtnMainMenue);
(*=====================================================================*)
FB_BtnTree(Zoom:='MANUAL_MAIN',
			deaktivieren:=FALSE,
			unsichtbar:=FALSE,
			Btn=> Visu.MainMenue.BtnManual);
	(*=====================================================================*)
	FB_BtnTree(Zoom:='MANUAL_ST00_0',
				deaktivieren:=FALSE,
				unsichtbar:=FALSE,
				Btn=> Visu.MainMenue.BtnManual_ST00_0);
			(*=====================================================================*)
	FB_BtnTree(Zoom:='MANUAL_ST00_1',
				deaktivieren:=FALSE,
				unsichtbar:=	FALSE,
				Btn=> Visu.MainMenue.BtnManual_ST00_1);
	FB_BtnTree(Zoom:='MANUAL_ST00_2',
				deaktivieren:=FALSE,
				unsichtbar:=						gTypeCode<>312  AND gTypeCode <> 4991,
				Btn=> Visu.MainMenue.BtnManual_ST00_2);
	(*=====================================================================*)
	FB_BtnTree(Zoom:='MANUAL_ST02_0',
				deaktivieren:=FALSE,
				unsichtbar:=						gTypeCode<>312  AND gTypeCode <> 4991,
				Btn=> Visu.MainMenue.BtnManual_ST02_0);
	(*=====================================================================*)
	FB_BtnTree(Zoom:='MANUAL_ST03_0',
				deaktivieren:=FALSE,
				unsichtbar:=FALSE,
				Btn=> Visu.MainMenue.BtnManual_ST03_0);
		(*=====================================================================*)
		(*Visu Seiten abhängig vom Stecker zuweisen*)
		CASE  gTypeCode OF
			312,4991:	FB_BtnTree.Zoom:='MANUAL_ST03_2';		(*93pol, 102pol*)
			322:		FB_BtnTree.Zoom:='MANUAL_ST03_3';		(*160pol*)
			4871:	FB_BtnTree.Zoom:='MANUAL_ST03_4';		(*154pol*)
			4872:	FB_BtnTree.Zoom:='MANUAL_ST03_5';		(*154 Rasterplatte*)
			522:		FB_BtnTree.Zoom:='MANUAL_ST03_6';		(*206pol*)
			550:		FB_BtnTree.Zoom:='MANUAL_ST03_8';		(*92pol*)
			564:		FB_BtnTree.Zoom:='MANUAL_ST03_7';		(*124pol*)
			569:		FB_BtnTree.Zoom:='MANUAL_ST03_9';		(*46pol*)
			5632,5633:	FB_BtnTree.Zoom:='MANUAL_ST03_10';		(*NOX5 NOX6*)
			5631:	FB_BtnTree.Zoom:='MANUAL_ST03_11';		(*NOX4*)
			5731:	FB_BtnTree.Zoom:='MANUAL_ST03_12';		(*88pol*)
			575,5753,5754,5755:		FB_BtnTree.Zoom:='MANUAL_ST03_13';		(*7pol,9pol,6pol,9pol*)
			5732:	FB_BtnTree.Zoom:='MANUAL_ST03_14';		(*88pol AMG*)
			5771:	FB_BtnTree.Zoom:='MANUAL_ST03_15';		(*120pol*)
			5772:	FB_BtnTree.Zoom:='MANUAL_ST03_16';		(*21pol*)
			580:		FB_BtnTree.Zoom:='MANUAL_ST03_17';		(*191pol*)
			5831:	FB_BtnTree.Zoom:='MANUAL_ST03_19';		(*72pol*)
			5832:	FB_BtnTree.Zoom:='MANUAL_ST03_18';		(*48pol*)
			5841,4993:	FB_BtnTree.Zoom:='MANUAL_ST03_20';		(*268pol, 102pol neu*)
			5842:	FB_BtnTree.Zoom:='MANUAL_ST03_21';		(*268polRT*)
			598:	FB_BtnTree.Zoom:='MANUAL_ST03_22';		(*33pol*)

		ELSE
			FB_BtnTree.Zoom:='MANUAL_ST03_1';					(*74,91,168,35 pol*)
		END_CASE
		FB_BtnTree(
					deaktivieren:=FALSE,
					unsichtbar:=FALSE,
					Btn=> Visu.MainMenue.BtnManual_ST03_xx);
		(*=====================================================================*)
		(*Visu Seiten abhängig vom Stecker zuweisen (nur eintragen wenn eine zweite Seite benötigt wird)*)
		FB_BtnTree.unsichtbar:=	FALSE;
		CASE  gTypeCode OF
			322:		FB_BtnTree.Zoom:='MANUAL_ST03_3_2';	(*160pol*)
			569:		FB_BtnTree.Zoom:='MANUAL_ST03_9_2';	(*46pol*)
			575,5753,5754,5755:		FB_BtnTree.Zoom:='MANUAL_ST03_13_2';(*7pol,9pol,6pol,9pol*)
			5633:	FB_BtnTree.Zoom:='MANUAL_ST03_10_2';		(*NOX5 NOX6*)
(*			5841,4993:	FB_BtnTree.Zoom:='MANUAL_ST03_20_2';	*)	(*268pol, 102pol neu*)
			5842:	FB_BtnTree.Zoom:='MANUAL_ST03_21_2';	(*268polRT*)

		ELSE
			FB_BtnTree.unsichtbar:=	TRUE;
		END_CASE
		FB_BtnTree(
					deaktivieren:=FALSE,
					Btn=> Visu.MainMenue.BtnManual_ST03_xx_2);
	(*=====================================================================*)
	FB_BtnTree(	Zoom:='MANUAL_ST08_0',
				deaktivieren:=FALSE,
				unsichtbar:=FALSE,
				Btn=> Visu.MainMenue.BtnManual_ST08_0);
			(*=====================================================================*)
			FB_BtnTree(Zoom:='MANUAL_ST08_1',
						deaktivieren:=FALSE,
						unsichtbar:=FALSE,
						Btn=> Visu.MainMenue.BtnManual_ST08_1);
			(*=====================================================================*)
			FB_BtnTree(Zoom:='MANUAL_ST08_2',
						deaktivieren:=FALSE,
						unsichtbar:=FALSE,
						Btn=> Visu.MainMenue.BtnManual_ST08_2);
			(*=====================================================================*)
			FB_BtnTree(Zoom:='MANUAL_ST08_3',
						deaktivieren:=FALSE,
						unsichtbar:=FALSE,
						Btn=> Visu.MainMenue.BtnManual_ST08_3);
			(*=====================================================================*)
			FB_BtnTree(Zoom:='MANUAL_ST08_4',
						deaktivieren:=FALSE,
						unsichtbar:=FALSE,
						Btn=> Visu.MainMenue.BtnManual_ST08_4);
(*=====================================================================*)
FB_BtnTree(Zoom:='TD_MAIN',
			deaktivieren:=FALSE,
			unsichtbar:=FALSE,
			Btn=> Visu.MainMenue.BtnTD);
	(*=====================================================================*)
	FB_BtnTree(Zoom:='TD_01_EDIT',
				deaktivieren:=FALSE,
				unsichtbar:=FALSE,
				Btn=> Visu.MainMenue.BtnTD01_Edit);
	IF	FB_BtnTree.Zoom = CurrentVisu THEN
		str_CurrentVisu_TD:=FB_BtnTree.Zoom;
	 END_IF
	(*=====================================================================*)
	FB_BtnTree(Zoom:='TD_02_EDIT',
				deaktivieren:=FALSE,
				unsichtbar:=FALSE,
				Btn=> Visu.MainMenue.BtnTD02_Edit);
	IF	FB_BtnTree.Zoom = CurrentVisu THEN
		str_CurrentVisu_TD:=FB_BtnTree.Zoom;
	 END_IF
(*=====================================================================*)
FB_BtnTree(	Text:='MP_MAIN',
			Zoom:='MP_ST1',
			deaktivieren:=FALSE,
			unsichtbar:=FALSE,
			Btn=> Visu.MainMenue.BtnMP_Main);
	(*=====================================================================*)
	FB_BtnTree(Zoom:='MP_ST1',
			deaktivieren:=FALSE,
			unsichtbar:=FALSE,
			Btn=> Visu.MainMenue.BtnMP_ST1);
	(*=====================================================================*)
	FB_BtnTree(Zoom:='MP_ST2',
			deaktivieren:=FALSE,
			unsichtbar:=FALSE,
			Btn=> Visu.MainMenue.BtnMP_ST2);
	(*=====================================================================*)
	FB_BtnTree(Zoom:='MP_DATE',
				deaktivieren:=FALSE,
				unsichtbar:=FALSE,
				Btn=> Visu.MainMenue.BtnMP_Date);
	(*=====================================================================*)
	FB_BtnTree(Zoom:='MP_SERVICE',
				deaktivieren:=FALSE,
				unsichtbar:=FALSE,
				Btn=> Visu.MainMenue.BtnMP_Service);
(*=====================================================================*)
FB_BtnTree(Zoom:='SYSTEM_MAIN',
			deaktivieren:=FALSE,
			unsichtbar:=FALSE,
			Btn=> Visu.MainMenue.BtnSystem);
		(*=====================================================================*)
		FB_BtnTree(Zoom:='LOGFILE',
					deaktivieren:=FALSE,
					unsichtbar:=FALSE,
					Btn=> Visu.MainMenue.Btn_ErrorLog);
		(*Error Log wird mit vbs Skript gestartet*)
		NT_StartProcess(
			NETID:=,
			PATHSTR		:='C:\Windows\System32\wscript.exe',
			DIRNAME		:=s_tools_path,
			COMNDLINE	:='logfile.vbs',
			START			:=Visu.MainMenue.Btn_ErrorLog.tasten,
			TMOUT			:=T#10s);
		(*=====================================================================*)
		FB_BtnTree(Zoom:='SYSTEM_ERRORLIST',
					deaktivieren:=FALSE,
					unsichtbar:=FALSE,
					Btn=> Visu.MainMenue.Btn_ErrorList);
		(*=====================================================================*)
		FB_BtnTree(Zoom:='SYSTEM_GST',
					deaktivieren:=FALSE,
					unsichtbar:=FALSE,
					Btn=> Visu.MainMenue.Btn_Gst);
		(*=====================================================================*)
		FB_BtnTree(Zoom:='SYSTEM_STEP_DIAG',
			deaktivieren:=FALSE,
			unsichtbar:=FALSE,
			Btn=> Visu.MainMenue.Btn_Step_Diag);
		(*=====================================================================*)
		FB_BtnTree(Zoom:='SYSTEM_LNG',
					deaktivieren:=FALSE,
					unsichtbar:=FALSE,
					Btn=> Visu.MainMenue.Btn_Lng);
		(*=====================================================================*)
		FB_BtnTree(Zoom:='EXIT',
					deaktivieren:=FALSE,
					unsichtbar:=FALSE,
					Btn=> Visu.MainMenue.Btn_VisuBeenden);
END_ACTION

(* POU zLibrary/ept/MainMenue/FB_Btn, ST *)
FUNCTION_BLOCK FB_Btn
VAR_INPUT
	unsichtbar			: BOOL;
	deaktivieren		: BOOL;
	Zoom				: STRING(50);
	Text				: STRING(50);
END_VAR
VAR_OUTPUT
	Btn		:sButtonVisu_Tree;
END_VAR
VAR
END_VAR
IF 	Text = '' THEN
	Btn.Text:=Zoom;
ELSE
	Btn.Text:=Text;
END_IF
Text:='';
Btn.Zoom:=Zoom;
Btn.deaktivieren:=deaktivieren;
Btn.unsichtbar:=unsichtbar;

IF	Btn.Text = CurrentVisu THEN
	Btn.innenFarbe:=Color.darkgrey;
ELSE
	Btn.innenFarbe:=Color.lightgrey;
END_IF
IF	deaktivieren THEN
	Btn.Textfarbe:=Color.grey;
ELSE
	Btn.Textfarbe:=Color.black;
END_IF
END_FUNCTION_BLOCK

(* POU zLibrary/ept/ST_Path, ST *)
PROGRAM ST_Path
VAR_INPUT
	Start				: BOOL;
END_VAR
VAR_OUTPUT
	Done				: BOOL;
	Error_				: BOOL;
	nErrId				: UDINT;
END_VAR
VAR

	fb_state_entry		: ST_StateEntry;

	fb_xml_srv_read		: FB_XmlSrvReadByName;	(* XML Baustein zum Auslesen von Meldungen *)
	s_PLC_path_name		: T_MaxString;				(* Pfad füR XML Baustein *)

	len_str				: INT;
	mid_str				: STRING(1);

END_VAR
VAR_TEMP
	i					:INT;
END_VAR
(*======================================================
   FB: Start eines Win Prozess mit Prüfung 
 ------------------------------------------------------
   Auth: 		Werner Friedl   						 
   Date: 		06.03.2019   						     
   Rev.: 		1.0	
   Desc:		Mit diesem Programm wird der PLC Pfad und der Projektpfad sowie der PLC- Name eingelesen
		
		Achtung!
		unter 
			"Projekt => Optionen => TwinCAT "
			musse der Haken bei
			"Sympolbeschreibung als Datei herunterladen"
			gesetzt sein.

   Historie:   1.0

=======================================================*)
fb_state_entry(i16_pos:= 1);

CASE fb_state_entry.i16_step OF
(*=======================================================*)
INIT_OBJ:

	fb_state_entry.i16_next_step:=INIT;

(*=======================================================*)
INIT:  fb_state_entry.s_debugtext:='PLC Projektpfad mit Projektnamen aus TPY auslesen Achtung!! Bootprojekt muss erstellt sein';

	IF fb_state_entry.E THEN
		fb_xml_srv_read.sFilePath := 'C:\TwinCAT\Boot\CurrentPlc_1.tpy';
		fb_xml_srv_read.sXPath :='/PlcProjectInfo/ProjectInfo/Path';
		fb_xml_srv_read.sSymName := 'ST_Path.s_PLC_path_name';
		fb_xml_srv_read.bExecute := TRUE;
		Error_:=FALSE;
	END_IF

	(*-----------------------Weiterschaltbedingungen----------------------------*)
	IF fb_xml_srv_read.bBusy THEN
		fb_xml_srv_read.bExecute := FALSE;
		fb_state_entry.i16_next_step := 20;
	END_IF

(*=======================================================*)
20:  fb_state_entry.s_debugtext:='Lesevorgang erfolgreich?';

	(*-----------------------Weiterschaltbedingungen----------------------------*)
	IF  NOT fb_xml_srv_read.bBusy  THEN
		IF NOT fb_xml_srv_read.bError THEN
			fb_state_entry.i16_next_step := 30;
		ELSE	(* Fehler *)
			s_PLC_Path_name:='!!! not found !!!';
			nErrId := fb_xml_srv_read.nErrId;
			fb_state_entry.i16_next_step := BEREIT;
			Error_:= TRUE;
		END_IF
	END_IF

	(*PLC Name und Pfad trennen *)
	s_PLC_name:=s_PLC_path_name;
	s_PLC_name:=s_PLC_path_name;
	len_str:=LEN(s_PLC_path_name);
	i:=0;

	FOR i:=1 TO len_str DO
		s_PLC_name:=DELETE(s_PLC_name,FIND(s_PLC_name,'\'),1);
	END_FOR

	s_PLC_path:=s_PLC_path_name;
	s_PLC_path:=DELETE(s_PLC_Path,LEN(s_PLC_path)-FIND(s_PLC_path,s_PLC_name)+1,FIND(s_PLC_path,s_PLC_name));
	s_Projekt_path:=s_PLC_path;

	len_str:=LEN(s_Projekt_path);
	s_Projekt_path:=LEFT(s_Projekt_path, len_str-1);

	(*PLC-Pfad löschen*)
	mid_str:='';
	len_str:=LEN(s_Projekt_path);
	FOR i:=1 TO LEN(s_Projekt_path) DO
			IF		mid_str <> '\' THEN
					s_Projekt_path:=LEFT(s_Projekt_path, len_str-i);
					mid_str:=MID(s_Projekt_path, 1 , len_str-i);
			END_IF
	END_FOR
(*=======================================================*)
30:  fb_state_entry.s_debugtext:='Pfade zusammen bauen';

	IF	s_Projekt_path <> '' THEN
		fb_state_entry.i16_next_step := BEREIT;
	END_IF

	IF	fb_state_entry.X THEN
		IF	FIND(s_tools_path,':') = 0 THEN
			s_tools_path:=CONCAT(s_Projekt_path,s_tools_path);
		END_IF

		IF	FIND(s_ud_path,':') = 0 THEN
			s_ud_path:=CONCAT(s_Projekt_path,s_ud_path);
		END_IF

		IF	FIND(MP_TDPathLocal,':') = 0 THEN
			MP_TDPathLocal:=CONCAT(s_Projekt_path,MP_TDPathLocal);
		END_IF

		IF	FIND(MP_TDPathService,':') = 0 THEN
			MP_TDPathService:=CONCAT(s_Projekt_path,MP_TDPathService);
		END_IF

		IF	FIND(MP_LocalDriveRoot,':') = 0 THEN
			MP_LocalDriveRoot:=CONCAT(s_Projekt_path,MP_LocalDriveRoot);
		END_IF

		IF	FIND(MP_ExportDrive,':') = 0 THEN
			MP_ExportDrive:=LEFT(s_PLC_path_name, 2);
		END_IF

		IF	FIND(MP_ExportDrivePathTD,'_') = 0 THEN
			MP_ExportDrivePathTD:=CONCAT(s_Projekt_path,MP_ExportDrivePathTD);
		END_IF

		IF	FIND(MP_ExportDrivePathMP,'_') = 0 THEN
			MP_ExportDrivePathMP:=CONCAT(s_Projekt_path,MP_ExportDrivePathMP);
		END_IF

		IF	FIND(LOG_RDPathLocal,':') = 0 THEN
			LOG_RDPathLocal:=CONCAT(s_Projekt_path,LOG_RDPathLocal);
		END_IF

		IF	FIND(LOG_ExportDrivePathRD,'_') = 0 THEN
			LOG_ExportDrivePathRD:=CONCAT(s_Projekt_path,LOG_ExportDrivePathRD);
		END_IF

	END_IF

(*=======================================================*)
BEREIT:  fb_state_entry.s_debugtext:='Warten auf Start';

	IF	fb_state_entry.E THEN
		Start:= FALSE;
		Done := TRUE;
	END_IF

	IF	Start THEN
		fb_state_entry.i16_next_step:=INIT;
	END_IF

	IF	fb_state_entry.X THEN
		Done := FALSE;
		Error_:= FALSE;
	END_IF

END_CASE

fb_state_entry(i16_pos:= 2);
(*========================================================================================*)

(* XML *)
fb_xml_srv_read(
	sNetId:= '',
	ePath:= PATH_GENERIC,
	nMode:= XMLSRV_SKIPMISSING,
	sSymName:= ,
	sFilePath:= ,
	sXPath:= ,
	bExecute:= ,
	tTimeout:= t#10s,
	bBusy=> ,
	bError=> ,
	nErrId=> );
END_PROGRAM

(* POU zLibrary/ept/min_exit/ST_MinExit, ST *)
PROGRAM ST_MinExit
VAR
	btn_min					: sButtonVisu;
	btn_exit					: sButtonVisu;

	fb_f_trig_minimieren		: F_TRIG;
	fb_tof_minimieren			: TOF;
	NT_StartProcess 			: NT_StartProcess;
	s_comndline						:STRING(255);
END_VAR
(*
in der C:\TwinCAT\Plc\TwinCAT PLC Control.ini muss
NoFullScreenMode=No umgestellt werden
=====================================================================*)



btn_min.Text:='_';
btn_min.Enable:=FALSE;
IF	btn_min.Pressed THEN
	btn_min.BackgroundColor:=Color.darkgrey;
ELSE
	btn_min.BackgroundColor:=Color.lightgrey;
END_IF
btn_min.TextColor:=Color.black;
btn_min.Visible:=FALSE;
fb_f_trig_minimieren(CLK:=btn_min.Pressed);
fb_tof_minimieren(IN:=fb_f_trig_minimieren.Q,PT:=t#1s);

IF	fb_f_trig_minimieren.Q THEN
	NT_StartProcess.START:=TRUE;
END_IF
IF 	NT_StartProcess.BUSY THEN
	NT_StartProcess.START:=FALSE;
END_IF

		(*minimieren wird mit vbs Skript gestartet*)
	NT_StartProcess(
			NETID:=,
			PATHSTR	:='C:\Windows\System32\wscript.exe',
			DIRNAME	:=s_tools_path,
			COMNDLINE	:='minimieren.vbs',
			START		:=,
			TMOUT		:=T#10s);
(*=====================================================================*)
btn_exit.Text:='X';
btn_exit.Enable:=FALSE;
IF	btn_exit.Pressed THEN
	btn_exit.BackgroundColor:=Color.darkgrey;
ELSE
	btn_exit.BackgroundColor:=Color.lightgrey;
END_IF

btn_exit.TextColor:=Color.black;
btn_exit.Visible:=FALSE;
END_PROGRAM

(* POU zLibrary/ept/ST_SaveAndLoad, ST *)
PROGRAM ST_SaveAndLoad
VAR_OUTPUT
	st_ctrl_out			:struct_ctrl_out;
END_VAR
VAR
	b_init				:BOOL;
	fb_state_entry		:ST_StateEntry;
	fb_ton_quitt		:TON;

	NT_StartProcess 	:NT_StartProcess;
	fbFileDelete		:FB_FileDelete;

	s_script			:STRING;

	btn_load			:sButtonVisu;
	btn_save			:sButtonVisu;

END_VAR
VAR CONSTANT
		s_bbgenMachineToSrv				:STRING:=		'_TD_save.bat';
		s_bbgenSrvToMachine				:STRING:=		'_TD_load.bat';

END_VAR
(*======================================================
   ST_SaveAndLoad
 ------------------------------------------------------
   Auth: 		Werner Friedl   						 
   Date: 		06.10.2020   						     
   Rev.: 		1.0	
   Desc:		Die bat Datein zum laden und speichern der BBgen Dateien werden hier ausgeführt.
			mit der Constante b_wkzBereinigen kann bestimmt werden, ob die Werkzeugdateu vorher gelöscht wird.

 ========================================================*)
IF	NOT b_init THEN
	b_Init:=TRUE;
END_IF
CallPrg();
Btn_init();
(* ========================================================*)
fb_ton_quitt(IN:= , PT:= t#100ms, Q=> , ET=> );

fb_state_entry(i16_pos:= 1);
CASE fb_state_entry.i16_step OF
(*=======================================================*)
INIT_OBJ:
		fb_state_entry.i16_next_step := INIT;

(*=======================================================*)
INIT:
	fb_state_entry.i16_next_step := BEREIT;

(*=======================================================*)
BEREIT:	fb_state_entry.s_debugtext:='warte auf Taster Save oder Load';

	IF fb_state_entry.E THEN
		st_ctrl_out.b_bereit:=TRUE;
		NT_StartProcess.START:=FALSE;
	END_IF

	(*-----------------------Weiterschaltbedingungen----------------------------*)
	IF 	btn_load.Pressed THEN
		fb_state_entry.i16_next_step:=110;
		s_script:=CONCAT(CURRENTLANGUAGE,s_bbgenSrvToMachine);
	ELSIF
		btn_save.Pressed THEN
		s_script:=CONCAT(CURRENTLANGUAGE,s_bbgenMachineToSrv);
		fb_state_entry.i16_next_step:=110;
	END_IF


	IF fb_state_entry.X THEN
		st_ctrl_out.b_busy:=TRUE;
		st_ctrl_out.b_bereit := FALSE;
		st_ctrl_out.b_fertig := FALSE;
	END_IF

(*=======================================================*)
110:fb_state_entry.s_debugtext:='start bat Script "Laden der Dateien vom Server"';

	IF 	fb_state_entry.E THEN
		NT_StartProcess.START:=TRUE;
	END_IF

	(*-----------------------Weiterschaltbedingungen----------------------------*)
	IF 	NT_StartProcess.BUSY THEN
		fb_state_entry.i16_next_step:=120;
	END_IF

	IF 	fb_state_entry.X THEN
		NT_StartProcess.START:=FALSE;
	END_IF

(*=======================================================*)
120:fb_state_entry.s_debugtext:='Warten auf fertig';

	IF	NOT btn_load.Pressed AND
		NOT btn_save.Pressed  THEN
		IF 	NT_StartProcess.ERR THEN
			fb_state_entry.s_debugtext:=CONCAT(fb_state_entry.s_debugtext,' ERRID => ');
			fb_state_entry.s_debugtext:=CONCAT(fb_state_entry.s_debugtext,UDINT_TO_STRING(NT_StartProcess.ERRID));
			fb_state_entry.i16_next_step:=FEHLER;
		ELSIF
			NOT NT_StartProcess.BUSY AND
			NOT NT_StartProcess.ERR AND
			fb_state_entry.fb_ton_Step.ET>t#3000ms THEN
			st_ctrl_out.b_busy:=FALSE;
			st_ctrl_out.b_fertig := TRUE;
			fb_state_entry.i16_next_step:=BEREIT;
		END_IF
	END_IF

(*=======================================================*)
STOP, FEHLER:

	IF fb_state_entry.E THEN
		st_ctrl_out.b_fehler := fb_state_entry.i16_step = FEHLER;
		st_ctrl_out.b_gestoppt := fb_state_entry.i16_step = STOP;
		st_ctrl_out.b_busy:=FALSE;
	END_IF

	IF	fb_state_entry.fb_ton_Step.ET > t#1000ms THEN   (*Quittiert sich selbst*)
		fb_state_entry.i16_next_step:=INIT;
	END_IF

END_CASE

fb_state_entry(i16_pos:= 2 );
END_PROGRAM
ACTION Btn_init:
btn_load.Text:='loadSrv';
btn_load.Enable:=CurrentUserLevel >=6 AND ModeSelect.Mode<=MODE_MANUAL;
IF btn_load.Enable THEN
	btn_load.TextColor:=Color.black;
ELSE
	btn_load.TextColor:=Color.grey;
END_IF
btn_load.Visible:= TRUE;

IF	btn_load.Pressed THEN
	btn_load.BackgroundColor:=Color.grey;
ELSE
	btn_load.BackgroundColor:=Color.lightgrey;
END_IF



btn_save.Text:='saveSrv';
btn_save.Enable:=CurrentUserLevel >=6 AND ModeSelect.Mode<=MODE_MANUAL;
IF btn_save.Enable THEN
	btn_save.TextColor:=Color.black;
ELSE
	btn_save.TextColor:=Color.grey;
END_IF
btn_save.Visible:= TRUE;

IF	btn_save.Pressed THEN
	btn_save.BackgroundColor:=Color.grey;
ELSE
	btn_save.BackgroundColor:=Color.lightgrey;
END_IF
END_ACTION
ACTION CallPrg:
NT_StartProcess(
	NETID:='',
	PATHSTR		:='C:\Windows\System32\cmd.exe',
	DIRNAME		:=s_tools_path,
	COMNDLINE	:=CONCAT('/C start /b ', s_script),
	START			:=,
	TMOUT			:=DEFAULT_ADS_TIMEOUT);


fbFileDelete(
	sNetId:= ,
	sPathName:= , 
	ePath:= PATH_GENERIC,
	bExecute:= ,
	tTimeout:= t#1s );
END_ACTION

(* POU zLibrary/ept/BDE/ST_Hydra8, ST *)
PROGRAM ST_Hydra8
VAR
	fb_tof_produktion			: TOF;
	fb_r_trig_signal			: R_TRIG;

	a_signal_produktion				AT %Q* : BOOL;
	a_signal_gutteil				AT %Q* : BOOL;
	a_signal_schlechtteil			AT %Q* : BOOL;
	a_signal_reserve				AT %Q* : BOOL;
	a_Fehlerfeld					: DWORD := 0;
END_VAR
(* Zeiten *)
fb_tof_produktion(
				IN:= 	(fb_r_trig_signal.Q AND
				ModeSelect.Mode=MODE_AUTO_RUN) OR
				(ST02_S1_40K01.BitInToCheck),
				PT:= T#60s,
				Q=>  a_signal_produktion,
				ET=> );

(* Flanken *)
IF	ST_CPU.LNG =CZ THEN
	fb_r_trig_signal(	CLK:= Robot01.State = STATE_OK);
END_IF

st_Hydra8Data.bStatus[_PRODUKTION] := a_signal_produktion;
END_PROGRAM

(* POU zLibrary/ept/BDE/ST_ImportHydraString, ST *)
PROGRAM ST_ImportHydraString
VAR_INPUT
	s_Path				: T_MaxString;
	sDateiName			: STRING;
	tStartTime			: TIME := T#10S;
END_VAR
VAR
	fb_state_entry			: ST_StateEntry;
	fbFindFiles			: FB_EnumFindFileList;
	fbFindFilesEntry		: ST_FindFileEntry;
	fbFileOpen			: FB_FileOpen;
	fbFileGets			: FB_FileGets;
	fbFileClose			: FB_FileClose;
	fbFileDelete			: FB_FileDelete;
	HelpString			: T_MaxString;
	fb_ton_start			: TON;
	hFile				:UINT:=0;
	nErrIdOpen			:UDINT;
	nErrIdRead			:UDINT;
	nErrIdClose			:UDINT;
	nErrIdDelete			:UDINT;
	sFileName			:STRING;

	iHelp				: INT;

	(* Für Anzeige in Visu *)
	iProduktionssperre	: INT;	(* 0 = nicht aktiv, 1 = aktiv, 2 = Status ungültig *)
END_VAR
VAR_OUTPUT
	Ready						:BOOL;
	Busy						:BOOL;
	Done						:BOOL;
	Error						:BOOL;
END_VAR
VAR CONSTANT
	sDatumPrefix				: STRING := 'DAT=';
	sZeitPrefix				: STRING := 'ZEI=';
	sOutput					: STRING := 'OUT';
	sTrennzeichen			: STRING := '|';
END_VAR
(*======================================================
   ST: ST_Import_Hydra_String
 ------------------------------------------------------
   Auth: 	Thomas Vilgis    						 
   Date: 	02.02.2022    						     
   Rev.: 	1.0	
   Desc:		Es wird alle 10 Sekunden (Zeit im Aufruf einstellbar) eine Textdatei mit 8 Status Ausgänge von Hydra erstellt.
			TwinCAT liest diese Datei aus und löscht sie dann.
			Es gibt nur eine Zeile in der Textdatei.
			Der erste Ausgang ist für den Status der Produktionssperre.
			Ein OUT Status steht nur in der Datei, wenn es eine Änderung gegeben hat.	
				
			So sieht die Datei aus: (alles in einer Zeile)
			OUT1=0|OUT2=0|OUT3=0|OUT4=0|OUT5=0|
			OUT6=0|OUT7=0|OUT8=0|DAT=02.02.2021|ZEI=07:16:00

   Historie: 	1.0

 ========================================================*)



(* Zeiten *)
fb_ton_start(IN:= NOT fb_ton_start.Q, PT:= tStartTime, Q=>  , ET=> );


(* ======================================Schrittkette======================================== *)
fb_state_entry(i16_pos:= 1);

CASE fb_state_entry.i16_step OF
(*=======================================================*)
	INIT_OBJ: fb_state_entry.s_debugtext:='initialisieren';

		(*-----------------------Weiterschaltbedingungen----------------------------*)
		IF fb_state_entry.fb_ton_Step.ET >= T#5S THEN
			fb_state_entry.i16_next_step:=BEREIT;
		END_IF

(*=======================================================*)
	BEREIT: fb_state_entry.s_debugtext:='Start';

		IF fb_state_entry.E THEN
			Ready := TRUE;
		END_IF

		(*-----------------------Weiterschaltbedingungen----------------------------*)
		IF fb_ton_start.Q THEN
			Error := FALSE;
			Busy := TRUE;
			Ready := FALSE;
			Done := FALSE;
			fb_state_entry.i16_next_step:=110;
		END_IF
		
		IF fb_state_entry.X THEN
			sFileName:=CONCAT(s_Path,sDateiName);
		END_IF
		
(*=======================================================*)
	110: fb_state_entry.s_debugtext:='HelpString löschen';
	
		IF fb_state_entry.E THEN
			HelpString := '';
		END_IF

		(*-----------------------Weiterschaltbedingungen----------------------------*)
		fb_state_entry.i16_next_step:=120;

(*=======================================================*)
	120: fb_state_entry.s_debugtext:='Prüfe, ob Datei vorhanden ist';

		IF fb_state_entry.E THEN
			fbFindFiles.bExecute := TRUE;
		END_IF

		(*-----------------------Weiterschaltbedingungen----------------------------*)
		IF fbFindFiles.bBusy THEN
			fb_state_entry.i16_next_step:=130;
		END_IF

(*=======================================================*)
	130: fb_state_entry.s_debugtext:='Prüfe, ob Datei vorhanden ist';

		(*-----------------------Weiterschaltbedingungen----------------------------*)
		IF NOT fbFindFiles.bBusy THEN
			fbFindFiles.bExecute := FALSE;
			IF NOT fbFindFiles.bError THEN
				IF fbFindFiles.nFindFiles = 1 THEN
					fb_state_entry.i16_next_step:=140;
				ELSE
					fb_state_entry.i16_next_step:=240;	(* Datei nicht vorhanden >> Auswertung *)
				END_IF
			ELSE
				fb_state_entry.i16_next_step:=FEHLER;
			END_IF
		END_IF

(*=======================================================*)
	140: fb_state_entry.s_debugtext:='Datei öffnen';

		IF fb_state_entry.E THEN
		   	fbFileOpen.bExecute:=TRUE;
		END_IF

		(*-----------------------Weiterschaltbedingungen----------------------------*)
		IF fbFileOpen.bBusy THEN
			fb_state_entry.i16_next_step:=150;
		END_IF

(*=======================================================*)
	150: fb_state_entry.s_debugtext:='Datei öffnen';

		(*-----------------------Weiterschaltbedingungen----------------------------*)
		IF 	NOT fbFileOpen.bBusy THEN

			fbFileOpen.bExecute:=FALSE;
			IF 	fbFileOpen.bError THEN
				nErrIdOpen:=fbFileOpen.nErrId;
				fb_state_entry.i16_next_step:=200;
			ELSE
				hFile := fbFileOpen.hFile;	(* Sehr wichtig hFile für FileRead und Fileclose übergeben *)
				fb_state_entry.i16_next_step:=160;
			END_IF
		END_IF

(*=======================================================*)
	160: fb_state_entry.s_debugtext:='Datei auslesen';

		IF fb_state_entry.E THEN
			fbFileGets.bExecute:=TRUE;
		END_IF

		(*-----------------------Weiterschaltbedingungen----------------------------*)
		IF  fbFileGets.bBusy THEN
			fb_state_entry.i16_next_step:=170;
		END_IF

(*=======================================================*)
	170: fb_state_entry.s_debugtext:='Datei auslesen';

		(*-----------------------Weiterschaltbedingungen----------------------------*)
		IF 	NOT fbFileGets.bBusy THEN
			fbFileGets.bExecute:=FALSE;
			IF 	fbFileGets.bError THEN
				nErrIdRead:=fbFileGets.nErrId;
				fb_state_entry.i16_next_step:=200;
			ELSE
				HelpString := fbFileGets.sLine;
				fb_state_entry.i16_next_step:=200;
			END_IF
		END_IF

(*=======================================================*)
	200: fb_state_entry.s_debugtext:='Datei schließen';

		IF fb_state_entry.E THEN
			fbFileClose.bExecute:=TRUE;
		END_IF

		(*-----------------------Weiterschaltbedingungen----------------------------*)
		IF 	fbFileClose.bBusy THEN
			fb_state_entry.i16_next_step:=210;
		END_IF

(*=======================================================*)
	210: fb_state_entry.s_debugtext:='Datei schließen';

		(*-----------------------Weiterschaltbedingungen----------------------------*)
		IF NOT fbFileClose.bBusy THEN
			fbFileClose.bExecute:=FALSE;
			IF 	fbFileClose.bError THEN
				nErrIdClose:=fbFileClose.nErrId;
				fb_state_entry.i16_next_step:=FEHLER;
			ELSE
				hFile := 0;
				fb_state_entry.i16_next_step:=220;
			END_IF
		END_IF
		
(*=======================================================*)
	220: fb_state_entry.s_debugtext:='Datei löschen';

		IF fb_state_entry.E THEN
			fbFileDelete.bExecute:=TRUE;
		END_IF

		(*-----------------------Weiterschaltbedingungen----------------------------*)
		IF 	fbFileDelete.bBusy THEN
			fb_state_entry.i16_next_step:=230;
		END_IF

(*=======================================================*)
	230: fb_state_entry.s_debugtext:='Datei löschen';

		(*-----------------------Weiterschaltbedingungen----------------------------*)
		IF NOT fbFileDelete.bBusy THEN
			fbFileDelete.bExecute:=FALSE;
			IF 	fbFileDelete.bError THEN
				nErrIdDelete:=fbFileDelete.nErrId;
				fb_state_entry.i16_next_step:=FEHLER;
			ELSE
				fb_state_entry.i16_next_step:=240;
			END_IF
		END_IF

(* Falls die Auswertung der Datei für jede Anlage unterschiedlich ist,
sollte man die Auswertung in einem eigenen Baustein machen *)
(*=======================================================*)
	240: fb_state_entry.s_debugtext:='Auswertung, ob Produktionssperre aktiv ist';

		IF fb_state_entry.E THEN
			IF fbFindFiles.nFindFiles = 0 THEN	(* Datei war gar nicht vorhanden *)
				iProduktionssperre := 2;	(* Status ungültig *)
			ELSE
				(* Suche nach OUT1= *)
				iHelp := FIND(HelpString, CONCAT(sOutput, '1='));
				IF iHelp > 0 THEN
					IF MID(HelpString, 1, 6) = '0' THEN	(* an Stelle 6 steht 0 oder 1 *)
						iProduktionssperre := 0;	(* nicht aktiv *)
					ELSIF MID(HelpString, 1, 6) = '1' THEN	(* an Stelle 6 steht 0 oder 1 *)
						iProduktionssperre := 1;	(* aktiv *)
					END_IF
				END_IF
			END_IF
		END_IF

		(*-----------------------Weiterschaltbedingungen----------------------------*)
		Busy := FALSE;
		Done := TRUE;
		fb_state_entry.i16_next_step:=BEREIT;
		
	

(*=======================================================*)
	FEHLER:
		IF fb_state_entry.E THEN
			Error := TRUE;
		END_IF

		(*-----------------------Weiterschaltbedingungen----------------------------*)
		fb_state_entry.i16_next_step:=BEREIT;

END_CASE


fb_state_entry(i16_pos:= 2);


fbFindFiles(
	bExecute	:= ,
	sNetId		:= '',
	sPathName	:= sFileName,
	pFindList	:= ADR(fbFindFilesEntry),
	cbFindList	:= SIZEOF(fbFindFilesEntry),
	tTimeout	:= t#1s );

 fbFileOpen(
	sNetId:='',
	sPathName:= sFileName,
	nMode:=FOPEN_MODEREAD,
	ePath:=PATH_GENERIC,
	bExecute:= ,
	tTimeout:=T#1s,
	hFile=> );

fbFileGets(
	sNetId:= , 
	hFile:= hFile, 
	bExecute:= , 
	tTimeout:= , 
	bBusy=> , 
	bError=> , 
	nErrId=> , 
	sLine=> , 
	bEOF=> );

fbFileClose(
	sNetId:='',
	hFile:=hFile,
	bExecute:= ,
	tTimeout:=T#1S);
	
fbFileDelete(
	sNetId:= , 
	sPathName:= sFileName, 
	ePath:= PATH_GENERIC, 
	bExecute:= , 
	tTimeout:= , 
	bBusy=> , 
	bError=> , 
	nErrId=> );
END_PROGRAM

(* POU System/LoginDialog/ImpExp_UD, ST *)
PROGRAM ImpExp_UD
VAR_INPUT
	Start_write				:BOOL;
	Start_read				:BOOL;
	path					:STRING(255);
	filename					:STRING(255);
END_VAR
VAR
	b_init					:BOOL;
	fb_state_entry				:ST_StateEntry;

	fb_xml_srv_read			: FB_XmlSrvReadByName;
	fb_xml_srv_write			: FB_XmlSrvWriteByName;

	fb_rtrig_Start_read			:R_TRIG;
	fb_rtrig_Start_write_to_server:R_TRIG;
	fb_ton_init				:TON;
	fb_ton_wz				:TON;
	fb_ton_uez				:TON;

	bError					: BOOL;
	nErrId					: UDINT;
	s_info					: STRING;
	MsgOK					: BOOL;
	MsgID					:STRING(20);

	UserList_Copy			: ARRAY [1..NO_OF_USERS] OF sUserData;

END_VAR

VAR_OUTPUT
	Busy					:BOOL;
	Done					:BOOL;
	Error					:BOOL;
	ErrorMsg				:STRING(255);
END_VAR

VAR CONSTANT
	SymName				:STRING:='.UD';
	xPath					:STRING:='/UD';
END_VAR

VAR_IN_OUT

END_VAR
(*======================================================
   PRG: XML Import und Export der UD
 ------------------------------------------------------
   Auth: 		Werner Friedl    						 
   Date: 		05.01.2021  						     
   Rev.: 		1.0	
   Desc:		
	- Userdate werden beim Neustart eingelesen
	- bei einer Änderung wird Änderung automatisch in die xml eingeragen

   Historie:   1.0

 ========================================================*)
fb_ton_init(IN:= TRUE, PT:=t#1500ms , Q=> , ET=> );
IF	NOT b_init AND fb_ton_init.Q THEN
	Start_read := TRUE;
	b_Init:=TRUE;
END_IF

(* ========================================================*)
fb_rtrig_Start_read();
IF	fb_rtrig_Start_read.Q AND
	NOT Start_write THEN
	Start_read:=TRUE;
END_IF

IF 	(MEMCMP(ADR(UserList_Copy),ADR(UD.UserList),SIZEOF(UserList_Copy))<>0)AND (*automatisch speichern im Manualmode*)
     	ModeSelect.Mode <=MODE_MANUAL AND
	NOT Start_read AND
	b_Init THEN
	Start_write := TRUE;
END_IF

(* ========================================================*)
fb_ton_wz(IN:= , PT:=t#3000ms , Q=> , ET=> );
IF	fb_ton_wz.Q THEN
	fb_ton_wz.IN:=FALSE;
	s_info := '';
END_IF

fb_state_entry(i16_pos:= 1);
CASE fb_state_entry.i16_step OF

(*=======================================================*)
0:	(*initialisieren*)
	Start_write := FALSE;
	Start_read := FALSE;
	fb_state_entry.i16_next_step:=BEREIT;

(*=======================================================*)
BEREIT: fb_state_entry.s_debugtext:='warte auf start';

	IF	Start_read THEN
		fb_state_entry.i16_next_step:=110;
	END_IF

	IF	Start_write THEN
		fb_state_entry.i16_next_step:=200;
	END_IF

	IF fb_state_entry.X THEN
		fb_ton_uez.IN:=FALSE;
		Start_write:=FALSE;
		Start_read:=FALSE;
		Busy:=TRUE;
		Error:=FALSE;
		Done:=FALSE;
		nErrId:=0;
		ErrorMsg:='';
		MsgID:='';
	END_IF

(*=======================================================*)
110: fb_state_entry.s_debugtext:='XML auslesen';	 

	IF fb_state_entry.E THEN
		fb_xml_srv_read.sFilePath := CONCAT(path,filename);
		fb_xml_srv_read.sSymName:=SymName;
		fb_xml_srv_read.sXPath :=xPath;
		fb_xml_srv_read.bExecute := TRUE;
	END_IF

	IF fb_xml_srv_read.bBusy THEN
		fb_xml_srv_read.bExecute := FALSE;
		fb_state_entry.i16_next_step := 120;
	END_IF

(*=======================================================*)
120: fb_state_entry.s_debugtext:='Lesevorgang erfolgreich?';

	IF  NOT fb_xml_srv_read.bBusy  THEN
		IF NOT fb_xml_srv_read.bError THEN
			fb_state_entry.i16_next_step := 900;
		ELSE	(* Fehler *)
			nErrId := fb_xml_srv_read.nErrId;
			IF	nErrId =1804 THEN
				MsgID:='PM15';
				ErrorMsg:='Die Datei UD.xml ist nicht vorhanden';
				fb_state_entry.i16_next_step := 200;	(*Datei wird erstellt*)
			ELSE
				MsgID:='PM16';
				ErrorMsg:='Fehler beim Einlesen der UD.xml Datei';
				fb_state_entry.i16_next_step := FEHLER;
			END_IF
		END_IF
	END_IF

	IF fb_state_entry.X THEN
		fb_ton_wz.IN:=TRUE;
		s_info:=CONCAT('read ',filename);
	END_IF

(*=======================================================*)
200: fb_state_entry.s_debugtext:='XML schreiben';

	IF fb_state_entry.E THEN
		fb_xml_srv_write.sFilePath := CONCAT(path,filename);
		fb_xml_srv_write.sSymName:=SymName;
		fb_xml_srv_write.sXPath :=xPath;
		fb_xml_srv_write.bExecute := TRUE;
	END_IF

	IF fb_xml_srv_write.bBusy THEN
		fb_xml_srv_write.bExecute := FALSE;
		fb_state_entry.i16_next_step := 220;
	END_IF

(*=======================================================*)
220: fb_state_entry.s_debugtext:='Schreiben erfolgreich?';

	IF  NOT fb_xml_srv_write.bBusy  THEN
		IF NOT fb_xml_srv_write.bError THEN
			UserList_Copy := UD.UserList;
			fb_state_entry.i16_next_step := 900;
		ELSE	(* Fehler *)
			nErrId := fb_xml_srv_write.nErrId;
			MsgID:='PM17';
			ErrorMsg:='Fehler beim Schreiben der UD.xml';
			fb_state_entry.i16_next_step := FEHLER;
		END_IF
	END_IF

	IF fb_state_entry.X THEN
		fb_ton_wz.IN:=TRUE;
		fb_ton_uez.IN:=TRUE;		(*automatisch auf Server speichern*)
		s_info:=CONCAT('write ',filename);
	END_IF

(*=======================================================*)
900: fb_state_entry.s_debugtext:='Fertig';

	Busy:=FALSE;
	Done:=TRUE;
	fb_state_entry.i16_next_step:=0;

(*=======================================================*)
FEHLER:

	IF fb_state_entry.E THEN
		MessageHandler.ClearMessageLines(sVisu:=Visu.Message);
	END_IF
	MessageHandler.Msg.ID:=MsgID;
	MessageHandler.Msg.Name:=ErrorMsg;
	MessageHandler.Msg.Text:=ErrorMsg;
	MessageHandler.Msg.Color:=Color.red;
	MessageHandler.Msg.Station:=0;

	MessageHandler(
		Prio:=2, 							(*1=highest, .. , 4=lowest*)
		Btn1Addr:=ADR(MsgOk),			(*Address of Button1 , if Zero then Button is unvisible*)
		Btn2Addr:=,						(*Address of Button2 , if Zero then Button is unvisible*)
		sVisu:=Visu.Message);

	IF MsgOK THEN
		MsgOk:=FALSE;
		fb_state_entry.i16_next_step:=0;
		Busy:=FALSE;
		Error:=TRUE;
	END_IF
END_CASE

fb_state_entry(i16_pos:= 2);


fb_xml_srv_read(
	sNetId:= '',
	ePath:= PATH_GENERIC,
	nMode:= XMLSRV_SKIPMISSING,
	sSymName:= ,
	sFilePath:= ,
	sXPath:= ,
	bExecute:= ,
	tTimeout:= t#10s,
	bBusy=> ,
	bError=> ,
	nErrId=> );

fb_xml_srv_write(
	sNetId:= '',
	ePath:= PATH_GENERIC,
	nMode:= XMLSRV_ADDMISSING,
	sSymName:=  ,
	sFilePath:= ,
	sXPath:= ,
	bExecute:= ,
	tTimeout:= t#10s,
	bBusy=> ,
	bError=> ,
	nErrId=> );


(*automatisch auf Server speichern=============================================*)
fb_ton_uez(PT:=t#20s);
fb_rtrig_Start_write_to_server(CLK:=fb_ton_uez.Q , Q=> );
(*
NT_StartProcess(
	NETID:='',
	PATHSTR	:='C:\Windows\System32\cmd.exe',
	DIRNAME	:='D:\Tools ',
	COMNDLINE	:='/C copy C:\MP\MachPara.xml \\10.16.50.9\bbgen\UML3\MD & @ping localhost -n 4 >NUL',
	START		:=fb_rtrig_Start_write_to_server.Q,
	TMOUT		:=t#10s);
*)
(*
NT_StartProcess(
	NETID:='',
	PATHSTR	:='C:\Windows\System32\wscript.exe',
	DIRNAME	:='D:\Tools',
	COMNDLINE	:='de_PD_aktuell_von_uml_nach_server.vbs',
	START		:=fb_rtrig_Start_write_to_server.Q,
	TMOUT		:=t#10s);
*)
END_PROGRAM

(* POU System/LoginDialog/UserLoginHandler, ST *)
PROGRAM UserLoginHandler
VAR
	Keypad								: UserLoginKeypad;
	btn_Login							: VisuButton;
	btn_LogOut							: VisuButton;
	btn_ChangeUserData				: VisuButton;
	btn_ChangePassword				: VisuButton;

	PasswordChangeActive				: BOOL;

	UserListIndexFixed					: INT;
	FixUserList							: BOOL;
	FP_FixUserList						: R_TRIG;
	FP_PasswordChangeActive			: R_TRIG;

	SelectedUser						: sUserData;
	UserLoggedOut						: sUserData;
	EmptyUser							: sUserData;

	CurrentVisuOld						: STRING;
	UserListIndexOld					: INT;

	InfoLogin              					: ErrorStruct;
	InfoLogout           					: ErrorStruct;

	TP_LogegdIn						: TP;
	TP_LogegdOut						: TP;

	Index								: INT;

	ton_AutoLoggedOut					: TON;
	b_Button							: BOOL;
	CopyCurrentVisu						: STRING;
	s_AutoLoggedOut					: STRING;

END_VAR
VAR_IN_OUT
	sVisu								: sVisuLoginDialog;
	UserList								: ARRAY [1..NO_OF_USERS] OF sUserData;

END_VAR
VAR_OUTPUT
	CurrentUser							: sUserData;
	UserLoggedIn						: BOOL;
END_VAR
(* Fix Administrator and Operator *)
UserList[1].UserName							:= 'Administrator';
(*UserList[1].UserPassword						:= '123';*)			(*PW in der ".....\UD\UserList.xml  " ändern und PLC neu starten*)
UserList[1].UserLevel							:= 7;
UserList[1].UserCanChangeOwnPassword			:= FALSE;

UserList[2].UserName							:= 'Service';
UserList[2].UserLevel							:= 6;
UserList[2].UserCanChangeOwnPassword			:= FALSE;

(* Fix UserLoggedOut *)
UserLoggedOut.UserName						:= 'Produktion';(*'Logged out';*)
UserLoggedOut.UserPassword					:= '';
UserLoggedOut.UserLevel						:= 1;
UserLoggedOut.UserCanChangeOwnPassword	:= FALSE;



Keypad(sVisu:= sVisu.LoginKeyPad,HidePasswordString:=NOT PasswordChangeActive);

FixUserList:= Keypad.Visible OR
			(CurrentUser.UserName<>UserLoggedOut.UserName AND CurrentUserLevel<6);

FP_FixUserList(CLK:= FixUserList );


(* Save Selecte UserIndex from Visu *)
IF 	FP_FixUserList.Q THEN
	UserListIndexFixed:=sVisu.UserListIndex;
END_IF;

(* Disable Selection in sVisu  *)
IF 	FixUserList THEN
	sVisu.UserListIndex:=UserListIndexFixed;
ELSE
	IF	sVisu.UserListIndex > 0 THEN
		SelectedUser:=UserList[sVisu.UserListIndex];
	END_IF
END_IF


(* Handle Keypad *)
FP_PasswordChangeActive(CLK:= PasswordChangeActive);
IF 	btn_Login.PressedFlag AND SelectedUser.UserPassword<>'' OR	(*Login with PW*)
	FP_PasswordChangeActive.Q THEN								(*PW-Change*)
	Keypad.Visible:=TRUE;
END_IF

IF 	Keypad.btnESC OR Keypad.btnOK OR CurrentVisuOld<>CurrentVisu THEN
	Keypad.Visible:=FALSE;
END_IF


(* Handle Login / Logout *)
btn_Login	(TextOn:= 'Login',	Button:= sVisu.btn_Login );
btn_LogOut	(TextOn:= 'Logout',	Button:= sVisu.btn_LogOut );

btn_Login.Enable:=TRUE;

btn_LogOut.Enable:=CurrentUser.UserName<>UserLoggedOut.UserName AND NOT PasswordChangeActive;


IF btn_LogOut.PressedFlag THEN
	(* Generate information Errorlog *)
	InfoLogout.Text			:=  CONCAT('LoginHandler: User ausgeloggt:',CurrentUser.UserName);
	InfoLogout.Typ			:=  2;
	InfoLogout.No			:=  1;
	InfoLogout.DateTime	:=  gVarDTSystemtime;
	TP_LogegdOut.IN		:= TRUE;

	CurrentUserLevel		:= 0;
	CurrentUser				:= UserLoggedOut;
END_IF

(*LogIn finished ok*)
IF 	Keypad.btnOK AND Keypad.InputString=SelectedUser.UserPassword AND NOT PasswordChangeActive OR		(*Login with PW, and PW ok*)
	btn_Login.PressedFlag AND SelectedUser.UserPassword='' THEN												(*Login without PW*)
	CurrentUserLevel		:= SelectedUser.UserLevel;
	CurrentUser				:= SelectedUser;
	(* Generate information Errorlog *)
	InfoLogin.Text			:= CONCAT('LoginHandler: User eingeloggt:',CurrentUser.UserName);
	InfoLogin.Typ			:= 2;
	InfoLogin.No			:= 1;
	InfoLogin.DateTime		:= gVarDTSystemtime;
	TP_LogegdIn.IN			:= TRUE;
END_IF


(* Edit Userlist *)

(* Show Edit Fields *)
sVisu.ShowEditFields:=(sVisu.UserListIndex>=2 AND CurrentUserLevel=7) OR (sVisu.UserListIndex>=3 AND CurrentUserLevel=6);

btn_ChangeUserData(Button:= sVisu.btn_ChangeUserData );
btn_ChangeUserData.Visible:=sVisu.ShowEditFields;

IF 	sVisu.UserEdit.UserName='' THEN
	btn_ChangeUserData.TextOn:= 'ChangeUserDataDel';
ELSE
	btn_ChangeUserData.TextOn:= 'ChangeUserData';
END_IF

IF 	btn_ChangeUserData.PressedFlag THEN
	(* Take new Userdatas when Username is not Administrator and Produktion *)
	IF 	sVisu.UserEdit.UserName <> 'Administrator' AND sVisu.UserEdit.UserName <> 'Produktion' THEN
		UserList[sVisu.UserListIndex]:=sVisu.UserEdit;
		IF 	UserList[sVisu.UserListIndex].UserName=''  THEN
			FOR index:= sVisu.UserListIndex TO DINT_TO_INT(NO_OF_USERS-1) BY 1 DO
				UserList[index]:=UserList[index+1];
			END_FOR
				UserList[index]:=EmptyUser;
		END_IF
	END_IF
END_IF

IF UserListIndexOld<>sVisu.UserListIndex
THEN
sVisu.UserEdit:=UserList[sVisu.UserListIndex];
END_IF

(* Change own Password from Allowed User *)
btn_ChangePassword(TextOn:= 'Passwortändern',Button:= sVisu.btn_ChangePassword );
btn_ChangePassword.Visible:=CurrentUser.UserCanChangeOwnPassword AND CurrentUser.UserName=SelectedUser.UserName;

IF 	btn_ChangePassword.PressedFlag THEN
	PasswordChangeActive:=TRUE;
END_IF

IF 	PasswordChangeActive	AND
	(Keypad.btnESC OR Keypad.btnOK OR CurrentVisuOld<>CurrentVisu) THEN
	IF Keypad.btnOK THEN
		UserList[sVisu.UserListIndex].UserPassword:=Keypad.InputString;
	END_IF
	PasswordChangeActive:=FALSE;
	Keypad.Visible:=FALSE;
END_IF

(* Compare Userleve with CurrentUser *)
IF 	CurrentUserLevel <> CurrentUser.UserLevel THEN
	CurrentUserLevel := CurrentUser.UserLevel;
END_IF

(* Check Current Username not Empty *)
IF  	CurrentUser.UserName = '' THEN
	CurrentUser := UserLoggedOut;
END_IF


UserLoggedIn:= (CurrentUser.UserName <> UserLoggedOut.UserName);


(* Last Operation!!!! *)
UserListIndexOld:=sVisu.UserListIndex;
CurrentVisuOld:=CurrentVisu;

IF 	TP_LogegdIn.Q THEN
	ErrorHandler.AddError(ErrorToAdd:=InfoLogin,sVisu:=Visu.ErrorHandler);
END_IF

IF 	TP_LogegdOut.Q THEN
	ErrorHandler.AddError(ErrorToAdd:=InfoLogout,sVisu:=Visu.ErrorHandler);
END_IF

TP_LogegdIn(PT:= t#1s );
TP_LogegdOut(PT:= t#1s );

TP_LogegdIn.IN:=FALSE;
TP_LogegdOut.IN:=FALSE;

(*========Benutzer automatisch abmelden=================================*)

b_Button:=
	Visu.ModeSelect.BtnManual.Pressed OR
	Visu.ModeSelect.BtnAuto.Pressed OR
	Visu.ModeSelect.BtnAutoStart.Pressed OR
	Visu.ModeSelect.BtnAutoStop.Pressed OR
	Visu.ModeSelect.BtnSpecial.Pressed OR
	Visu.ModeSelect.BtnRunEmpty.Pressed OR
	Visu.ModeSelect.BtnStepCycle.Pressed OR
	Visu.ModeSelect.BtnSpecial.Pressed OR
	Visu.ModeSelect.BtnSpecStep.Pressed OR
	Visu.ModeSelect.BtnHomeRun.Pressed OR
	Visu.ModeSelect.BtnReset.Pressed;

IF	CurrentVisu<>CopyCurrentVisu THEN
	b_Button:=TRUE;
	CopyCurrentVisu:=CurrentVisu;
END_IF

IF	CurrentUser.UserName<>UserLoggedOut.UserName AND
	MP.ST00.MaxLogInTime <> 0 THEN

	ton_AutoLoggedOut(
			IN:=NOT  b_Button,
			PT:=DINT_TO_TIME(MP.ST00.MaxLogInTime*60000) ,
			Q=> ,
			ET=> );
	s_AutoLoggedOut:=ET_TO_STRING(ton_AutoLoggedOut.PT - ton_AutoLoggedOut.ET);
	s_AutoLoggedOut:=LEFT(s_AutoLoggedOut,FIND( s_AutoLoggedOut,'s'));

	IF	ton_AutoLoggedOut.Q THEN
		(* Generate information Errorlog *)
		InfoLogout.Text                 := CONCAT('LoginHandler: User ausgeloggt:',CurrentUser.UserName);
		InfoLogout.Typ                  := 2;
		InfoLogout.No                   := 1;
		InfoLogout.DateTime         := gVarDTSystemtime;
		TP_LogegdOut.IN:=TRUE;

		CurrentUserLevel		:=1;
		CurrentUser				:=UserLoggedOut;
	END_IF

ELSE
	ton_AutoLoggedOut(IN:=FALSE);
	s_AutoLoggedOut:='';
END_IF
END_PROGRAM

(* POU System/LoginDialog/UserLoginKeypad, ST *)
FUNCTION_BLOCK UserLoginKeypad
VAR
	btn_Key1					: VisuButton;
	btn_Key2					: VisuButton;
	btn_Key3					: VisuButton;
	btn_Key4					: VisuButton;
	btn_Key5					: VisuButton;
	btn_Key6					: VisuButton;
	btn_Key7					: VisuButton;
	btn_Key8					: VisuButton;
	btn_Key9					: VisuButton;
	btn_Key0					: VisuButton;
	btn_KeyDot				: VisuButton;

	btn_KeyBack				: VisuButton;
	btn_KeyEsc				: VisuButton;
	btn_KeyClear			: VisuButton;
	btn_KeyOK					: VisuButton;
	btn_KeyVorzeichen	: VisuButton;

	InputStringLen		: INT;
	I									: INT;

	FP_Init						:	R_TRIG;
END_VAR
VAR_IN_OUT
	sVisu							: sNumericKeypad;
END_VAR
VAR_INPUT
	Visible						:	BOOL;
	HidePasswordString: BOOL;
END_VAR
VAR_OUTPUT
	InputString				:	STRING;
	btnOK							:	BOOL;
	btnESC						:	BOOL;
END_VAR
btn_Key0(	TextOn:= '0',	Button:= sVisu.btn_Key0 );
btn_Key1(	TextOn:= '1',	Button:= sVisu.btn_Key1 );
btn_Key2(	TextOn:= '2',	Button:= sVisu.btn_Key2 );
btn_Key3(	TextOn:= '3',	Button:= sVisu.btn_Key3 );
btn_Key4(	TextOn:= '4',	Button:= sVisu.btn_Key4 );
btn_Key5(	TextOn:= '5',	Button:= sVisu.btn_Key5 );
btn_Key6(	TextOn:= '6',	Button:= sVisu.btn_Key6 );
btn_Key7(	TextOn:= '7',	Button:= sVisu.btn_Key7 );
btn_Key8(	TextOn:= '8',	Button:= sVisu.btn_Key8 );
btn_Key9(	TextOn:= '9',	Button:= sVisu.btn_Key9 );
btn_KeyBack(	TextOn:= 'Back',	Button:= sVisu.btn_KeyBack );
btn_KeyEsc(	TextOn:= 'Esc',	Button:= sVisu.btn_KeyEsc );
btn_KeyClear(	TextOn:= 'Clear',	Button:= sVisu.btn_KeyClear );
btn_KeyOK(	TextOn:= 'OK',	Button:= sVisu.btn_KeyOK );

btn_KeyDot(	TextOn:= '.',	Button:= sVisu.btn_KeyDot );
btn_KeyVorzeichen(	TextOn:= '+/-',	Button:= sVisu.btn_KeyVorzeichen );

btn_KeyDot.Enable:=FALSE;
btn_KeyVorzeichen.Enable:=FALSE;

svisu.Visible:=Visible;
svisu.Enable:=Visible;

(* initialize  *)
FP_Init(CLK:= Visible);

IF FP_Init.Q
THEN
	InputString:='';
END_IF


InputStringLen:=LEN(InputString);

IF btn_Key0.PressedFlag
THEN
	InputString:=CONCAT(InputString,'0');
END_IF
IF btn_Key1.PressedFlag
THEN
	InputString:=CONCAT(InputString,'1');
END_IF
IF btn_Key2.PressedFlag
THEN
	InputString:=CONCAT(InputString,'2');
END_IF
IF btn_Key3.PressedFlag
THEN
	InputString:=CONCAT(InputString,'3');
END_IF
IF btn_Key4.PressedFlag
THEN
	InputString:=CONCAT(InputString,'4');
END_IF
IF btn_Key5.PressedFlag
THEN
	InputString:=CONCAT(InputString,'5');
END_IF
IF btn_Key6.PressedFlag
THEN
	InputString:=CONCAT(InputString,'6');
END_IF
IF btn_Key7.PressedFlag
THEN
	InputString:=CONCAT(InputString,'7');
END_IF
IF btn_Key8.PressedFlag
THEN
	InputString:=CONCAT(InputString,'8');
END_IF
IF btn_Key9.PressedFlag
THEN
	InputString:=CONCAT(InputString,'9');
END_IF

IF btn_KeyBack.PressedFlag
THEN
	InputString:=LEFT(InputString,InputStringLen-1);
END_IF

IF btn_KeyClear.PressedFlag
THEN
	InputString:='';
END_IF

IF btn_KeyEsc.PressedFlag
THEN
	InputString:='';
END_IF

InputStringLen:=LEN(InputString);
svisu.InputString:='';

IF HidePasswordString
THEN

	FOR i:=1 TO InputStringLen DO
		svisu.InputString:=CONCAT(svisu.InputString,'*');
	END_FOR
ELSE
	svisu.InputString:=InputString;
END_IF
btnOK:=btn_KeyOK.PressedFlag;
btnESC:=btn_KeyEsc.PressedFlag;
END_FUNCTION_BLOCK

(* POU System/TDHandler/TDHandler, ST *)
PROGRAM TDHandler
VAR

	WriteXML					: FB_XmlSrvWriteByName;
	ReadXML					: FB_XmlSrvReadByName;
	DeleteXML					: FB_FileDelete;
	DeleteXMLactive			: BOOL;

	FindFiles					: FB_EnumFindFileList;

	filesList						: ARRAY[1..NO_OF_FILES] OF ST_FindFileEntry;

	i,j							: DINT;

	FileNameWrite				: STRING(255);
	FileNameRead				: STRING(255);
	FileNameDelete				: STRING(255);

	FileWriteSource				: STRING(255);
	FileReadTarget				: STRING(255);


	FileNameSearch				: STRING(255);

	FileFilterOld					: STRING(255);
	FileIndexOld					: DINT;
	fb_rTrigFilList				: R_TRIG;

	BtnSaveAs					: VisuButton;
	BtnActivate					: VisuButton;
	BtnDelete					: VisuButton;

	FirstCycle					: BOOL;
	SetActivate					: BOOL := FALSE;

	Error						: ErrorStruct;
	ErrorElapsed				: R_TRIG;
	TDValid						: BOOL;
	FileNameReadCopy			: STRING(255);
	TDCopy						: sTypeData;
	TDempty					: sTypeData;
	TypeNameCopy				: STRING;
	fb_ExpActTDNo				: FB_ExporString;	(* Fehlermeldungen in Errorlog (txt) schreiben *)

	b_Dialog_save_as_on		: BOOL;

	s_Xpath						: T_MaxString;
	state						: INT:=0;
	s_Typecode					: T_MaxString;
	s_Typedescription			: T_MaxString;
	fb_TonDel					: TON;

END_VAR
VAR_IN_OUT
	sVisu : sTDHandler;
END_VAR
VAR_INPUT
	TDActivationAlowed			: BOOL; (* Typedata activation alowed *)
END_VAR
VAR_OUTPUT
	DownLoadTime				: STRING;
END_VAR
info();
DisableTD();
IF 	NOT FirstCycle THEN
	IF	MP.sLastTDfile <> '' AND
		MP_TDPathLocal <> '' THEN
		FileNameRead 		:= CONCAT(MP_TDPathLocal,MP.sLastTDfile);
		FileReadTarget		:= '.TD';
		s_Xpath:='/dataentry/TD';
		ReadXML.bExecute	:=TRUE;
		FirstCycle:=TRUE;
	END_IF
END_IF

IF TD.TypeName <> TypeNameCopy THEN
	TypeNameCopy:=TD.TypeName;
	fb_ExpActTDNo.Start:=TRUE;
	MP.ST02.Override_Band:=TD.Override_Band;
	MP.ST00.Override:=TD.Override_Robi;
END_IF

IF 	FIND(sVisu.FileFilter,'*')= 0 THEN
	sVisu.FileFilter:=CONCAT(sVisu.FileFilter,'*');
END_IF

FileNameSearch := CONCAT(MP_TDPathLocal,sVisu.FileFilter);
FileNameSearch := CONCAT(FileNameSearch,MP_TDFileExtension);

fb_rTrigFilList(CLK:=CurrentVisu = 'TD_MAIN' );
IF 	FileIndexOld <> sTDHandler.FileIndex OR
	fb_rTrigFilList.Q OR
	FileFilterOld<>sVisu.FileFilter  THEN
	FileIndexOld:= sTDHandler.FileIndex;
	sVisu.FileListUpdate:=TRUE;
	FileFilterOld:=sVisu.FileFilter;
END_IF


(* --------------------------------------------------------------- *)
(* ------------------ Function Calls --------------------- *)
(* --------------------------------------------------------------- *)

FindFiles(
	bExecute			:=sVisu.FileListUpdate,
	sNetId				:= '',
	sPathName			:= FileNameSearch,
	pFindList			:= ADR(filesList),
	cbFindList		:= SIZEOF(filesList) ,
	tTimeout			:= t#1s );

sVisu.FileListUpdate:=FALSE;

WriteXML(
	sNetId				:= '',
	nMode				:= XMLSRV_ADDMISSING,
	sSymName			:= FileWriteSource,
	sFilePath			:= FileNameWrite ,
	sXPath				:= '/dataentry/TD',
	tTimeout			:= t#10s
 );

IF 	NOT WriteXML.bBusy OR WriteXML.bError THEN

	IF 	WriteXML.bExecute THEN
		sVisu.FileListUpdate:=TRUE;
	END_IF
	WriteXML.bExecute:=FALSE;

END_IF

ReadXML(
	sNetId				:= '',
	nMode				:= XMLSRV_SKIPMISSING ,
	sSymName			:= FileReadTarget,
	sFilePath			:= FileNameRead,
	sXPath				:= s_Xpath,				(* '/dataentry/TD',*)
	tTimeout			:= t#15s
 );


IF 	NOT ReadXML.bBusy AND
	ReadXML.bExecute	 THEN
	IF	FileReadTarget = '.TD' AND
		FileNameRead <>'' THEN
		lastTDActivate:=FileNameRead;
	END_IF
	TDValid:=TRUE;
END_IF

IF 	NOT ReadXML.bBusy OR
	ReadXML.bError THEN
	ReadXML.bExecute:=FALSE;
END_IF

j:=1;
FOR i:=1 TO NO_OF_FILES DO
	IF 	filesList[i].sFileName<>'' THEN
		sVisu.FileList[j]:=filesList[i].sFileName;
		j:=j+1;
	ELSE
		sVisu.FileList[j]:='';
		j:=j+1;
	END_IF
END_FOR

(* --------------------------------------------------------------- *)
(* -----------------  Visu interface ----------------------------- *)
(* --------------------------------------------------------------- *)
IF 	sVisu.FileIndex = 0 THEN
	sVisu.FileIndex:=1;
END_IF
sVisu.FileNameSelected:=sVisu.FileList[sVisu.FileIndex];

BtnActivate(
	Enable			:= sVisu.FileNameSelected <> MP.sLastTDfile AND sVisu.FileNameSelected <>'' AND ModeSelect.Mode <= MODE_MANUAL,
	Visible			:= TRUE,
	TextOn			:= 'Activate',
	TextOff			:= 'Activate',
	Button			:= sVisu.BtnActivate
  );

IF 	BtnActivate.PressedFlag THEN
	TD:=TDempty;
	TDCopy:=TDempty;
	FileNameRead 		:= CONCAT(MP_TDPathLocal,sVisu.FileNameSelected);
	FileReadTarget		:= '.TD';
	ReadXML.bExecute	:=TRUE;
	SetActivate			:=TRUE;
	gTypeDataValid 		:= FALSE;
	s_Xpath:='/dataentry/TD';
	MP.sLastTDfile		:=sVisu.FileNameSelected;
END_IF


IF 	SetActivate AND
	ModeSelect.Mode <= MODE_MANUAL OR gTInfo_FirstStart THEN

	IF 	NOT ReadXML.bBusy AND NOT ReadXML.bError THEN
		DownLoadTime:=gVarStrSystemTime;
		SetActivate:=FALSE;
		gTypeDataValid:=TRUE;
	ELSIF
		ReadXML.bBusy AND ReadXML.bError THEN
		SetActivate:=FALSE;
	END_IF
ELSIF
	ModeSelect.Mode<>MODE_MANUAL THEN
	SetActivate:=FALSE;
	(*ST00_LoadTInfo.Start:=FALSE;*)
END_IF
sVisu.TypeDataValid:=gTypeDataValid;


(*Automatisch sichern*)
IF	(MEMCMP(ADR(TDCopy), ADR(TD), SIZEOF(TDCopy)) <> 0 ) AND
	lastTDActivate<> '' AND
	NOT ReadXML.bBusy AND
	NOT ReadXML.bError THEN
	FileNameWrite	:= lastTDActivate;
	FileWriteSource	:= '.TD';
	WriteXML.bExecute:=TRUE;
END_IF
TDCopy:=TD;
TD.TypeName	:= MP.sLastTDfile;

(*============================*)

BtnSaveAs(
	Enable			:= sVisu.FileNameSelected = MP.sLastTDfile AND CurrentUserLevel >=6,
	Visible			:= TRUE ,
	TextOn			:= 'SaveAs',
	TextOff			:= 'SaveAs',
	Button			:= sVisu.BtnSaveAs
  );

IF 	BtnSaveAs.PressedFlag THEN
	b_Dialog_save_as_on:=TRUE;
END_IF

IF 	sVisu.FileNameSaveAs <>'' THEN
	FileNameWrite	:= CONCAT(MP_TDPathLocal,sVisu.FileNameSaveAs);
	FileNameWrite	:= CONCAT(FileNameWrite,MP_TDFileExtension);
  	TD.TypeName	:= sVisu.FileNameSaveAs;

	FileWriteSource	:= '.TD';
	WriteXML.bExecute:=TRUE;

	sVisu.FileNameSaveAs:='';
	b_Dialog_save_as_on:=FALSE;

END_IF

BtnDelete(
	Enable			:= sVisu.FileNameSelected <> MP.sLastTDfile AND sVisu.FileNameSelected<>'' AND CurrentUserLevel >=6,
	Visible			:= TRUE ,
(*	Enable			:= sVisu.FileNameSelected<>'',
	Visible			:= sVisu.FileNameSelected<>'',*)
	TextOn			:= 'Del',
	TextOff			:= 'Del',
	Button			:= sVisu.BtnDelete
  );


IF 	BtnDelete.PressedFlag THEN
	FileNameDelete 		:= CONCAT(MP_TDPathLocal,sVisu.FileNameSelected);
	DeleteXML.bExecute:=TRUE;
END_IF

DeleteXML(
	sNetId			:= '',
	sPathName		:= FileNameDelete,
	tTimeout		:= t#10s
 );
IF 	DeleteXML.bExecute AND
	DeleteXML.bBusy THEN
	DeleteXMLactive:=TRUE;
END_IF

IF 	DeleteXMLactive AND
	(NOT DeleteXML.bBusy OR  DeleteXML.bError) THEN
	sVisu.FileListUpdate:=TRUE;
	DeleteXMLactive:=FALSE;
END_IF


DeleteXML.bExecute:=FALSE;

(*send to ErrorHandler (to show Error-Line and to add into ErrorLogFile) *)
IF 	NOT TDValid THEN
	ErrorElapsed(CLK:= Error.Text<>''AND gVarDTSystemtime<> ErrorHandler.EmptyError.DateTime);
	IF 	ErrorElapsed.Q THEN
		Error.DateTime:=
		gVarDTSystemtime;
	END_IF
	Error.Text	:= 'TD: NOT valid';
	Error.No		:= 1;
	Error.Typ	:= 0;			(* 0=red 1:=orange 2:=blue *)
	ErrorHandler.AddError
				(ErrorToAdd	:=Error,
				sVisu		:=Visu.ErrorHandler);
END_IF

IF	TDValid AND
	FileNameReadCopy<> FileNameRead THEN
	Error.Text		:= CONCAT('TD: open ',FileNameRead);
	Error.DateTime	:=gVarDTSystemtime;
	Error.No			:= 1;
	Error.Typ		:= 0;			(* 0=red 1:=orange 2:=blue *)
	ErrorHandler.AddError
				(ErrorToAdd	:=Error,
				sVisu		:=Visu.ErrorHandler);

	FileNameReadCopy:=FileNameRead;
END_IF

IF	TDValid AND
	WriteXML.bExecute THEN
	Error.Text		:= CONCAT('TD: save ',FileNameWrite);
	Error.DateTime	:=gVarDTSystemtime;
	Error.No			:= 1;
	Error.Typ		:= 0;			(* 0=red 1:=orange 2:=blue *)
	ErrorHandler.AddError
				(ErrorToAdd	:=Error,
				sVisu		:=Visu.ErrorHandler);

END_IF

fb_ExpActTDNo(
	Start:= ,
	ExportStr:=TypeNameCopy ,
	FileName:= 'ActTD.txt',
	Path:=  s_tools_path,
	Mode:=FOPEN_MODEWRITE,
	Busy=> ,
	Done=> ,
	Error=> ,
	ErrorMsg=> );
END_PROGRAM
ACTION DisableTD:
(* Sperre der Typdateneingabe *)
gDisableTD := FALSE;
IF 	CurrentUserLevel <6  OR
	ModeSelect.Mode >  MODE_MANUAL THEN
	gDisableTD := TRUE;
END_IF
END_ACTION
ACTION Info:
(*immer wenn ein neu Datei ausgewhält wird, dann wird die Beschreibung und der Projektcode ausgelesen*)
fb_TonDel(PT:=t#20s);

IF 	FileIndexOld <> sTDHandler.FileIndex THEN
	fb_TonDel.IN:=FALSE;
	state:=5;
END_IF


CASE state OF
0:
	IF	fb_TonDel.Q THEN
		fb_TonDel.IN:=FALSE;
		s_Typecode:='';
		s_Typedescription:='';
	END_IF

5:
	IF 	FileIndexOld = sTDHandler.FileIndex AND
		NOT FindFiles.bBusy THEN
		state:=10;
	END_IF

10:
	FileNameRead 		:= CONCAT(MP_TDPathLocal,filesList[FileIndexOld].sFileName);
	FileReadTarget		:= 'TDHandler.s_Typecode';
	s_Xpath				:='/dataentry/TD/TYPECODE';
	ReadXML.bExecute	:=TRUE;
	IF	ReadXML.bBusy THEN
		state:=20;
		ReadXML.bExecute	:=FALSE;
	END_IF

20:
	IF	NOT ReadXML.bBusy AND
		NOT ReadXML.bError THEN
		state:=30;
	END_IF

30:
	FileNameRead 		:= CONCAT(MP_TDPathLocal,sVisu.FileNameSelected);
	FileReadTarget		:= 'TDHandler.s_Typedescription';
	s_Xpath				:='/dataentry/TD/TYPEDESCRIPTION';
	ReadXML.bExecute	:=TRUE;
	IF	ReadXML.bBusy THEN
		ReadXML.bExecute	:=FALSE;
		state:=40;
	END_IF

40:
	IF	NOT ReadXML.bBusy AND
		NOT ReadXML.bError THEN
		state:=0;
		fb_TonDel.IN:=TRUE;
	END_IF
END_CASE
END_ACTION

(* POU zLibrary/ept/Funktionsbausteine/FB_ExporString, ST *)
FUNCTION_BLOCK FB_ExporString
VAR_INPUT
	Start				:BOOL;
	ExportStr			:STRING(255);
	FileName		:STRING(255);
	Path				:STRING(255);
	Mode			:DWORD;
END_VAR
VAR_OUTPUT
	Busy				:BOOL;
	Done				:BOOL;
	Error				:BOOL;
	ErrorMsg			:STRING(255);

END_VAR
VAR
	fb_state_entry		:ST_StateEntry;
	nErrId				:UDINT;

	fbFileOpen			:FB_FileOpen;
	fbFilePuts			:FB_FilePuts;
	fbFileClose			:FB_FileClose;

	hFile				:UINT;

END_VAR

VAR CONSTANT
	Zeilenumbruch		:STRING:='$R$N';
END_VAR
(*======================================================
   PRG: FB_ExportString
 ------------------------------------------------------
   Auth: 		Werner Friedl    						 
   Date: 		30.10.2014    						     
   Rev.: 		1.0	
   Desc:		
		
   Historie:   1.0

 ========================================================*)
fb_state_entry(i16_pos:= 1);

CASE fb_state_entry.i16_step OF

0:	(*Objekt initialisieren*)
	fb_state_entry.i16_next_step:=INIT;

10:	(*initialisieren*)
	fb_state_entry.i16_next_step:=BEREIT;

BEREIT:(*Start*)

	IF	Start THEN  (*initialisieren*)
		Start:=FALSE;
		Busy:=TRUE;
		Error:=FALSE;
		Done:=FALSE;
		nErrId:=0;
		ErrorMsg:='';
		fb_state_entry.i16_next_step:=110;

	END_IF

110: (*Datei erstellen*)

	FileName:=CONCAT(Path,FileName);

	fbFileOpen.sPathName:=FileName;
 	fbFileOpen.bExecute:=TRUE;

	IF 	NOT fbFileOpen.bBusy   THEN
		fb_state_entry.i16_next_step:=120;
	END_IF

120: (*Datei erstellen*)

	IF 	NOT fbFileOpen.bBusy THEN
		fbFileOpen.bExecute:=FALSE;
		IF 	fbFileOpen.bError THEN
			nErrId:=fbFileOpen.nErrId;
			fb_state_entry.i16_next_step:=FEHLER;
			ErrorMsg:='Fehler beim Öffnen der Datei';
		ELSE
			fb_state_entry.i16_next_step:=130;
		END_IF
	END_IF

130: (*String in Datei eintragen*)
	IF fb_state_entry.E THEN
		;
	END_IF

	fbFilePuts.sLine:=CONCAT(ExportStr,Zeilenumbruch);
	fbFilePuts.bExecute:=TRUE;

	IF  fbFilePuts.bBusy THEN
		fb_state_entry.i16_next_step:=140;
	END_IF

140: (*String in Datei eintragen*)

	IF 	NOT fbFilePuts.bBusy THEN
		fbFilePuts.bExecute:=FALSE;
		IF 	fbFilePuts.bError THEN
			nErrId:=fbFilePuts.nErrId;
			fb_state_entry.i16_next_step:=150;
			ErrorMsg:='Fehler beim String Eintragen in der Datei';
			Error:=TRUE;
		ELSE
			fb_state_entry.i16_next_step:=150;
		END_IF
	END_IF

150:(*Datei schließen*)

	fbFileClose.bExecute:=TRUE;
	IF 	fbFileClose.bBusy THEN
		fb_state_entry.i16_next_step:=160;
	END_IF

160:(*Datei schließen*)

	IF NOT fbFileClose.bBusy THEN
		fbFileClose.bExecute:=FALSE;
		IF 	fbFileClose.bError THEN
			nErrId:=fbFileClose.nErrId;
			ErrorMsg:='Fehler beim Schließen der Datei';
			Error:=TRUE;
		ELSE
			fb_state_entry.i16_next_step:=170;
		END_IF
	END_IF

	IF	Error THEN
		fb_state_entry.i16_next_step:=FEHLER;
	END_IF

170: (*fertig*)
	Busy:=FALSE;
	Done:=TRUE;
	fb_state_entry.i16_next_step:=10;

FEHLER: (*Fehler*)
	fb_state_entry.i16_next_step:=10;
	Busy:=FALSE;
	Error:=TRUE;
END_CASE

fb_state_entry(i16_pos:= 2 );

fbFileOpen(
	sNetId:='',
	sPathName:= ,
	nMode:=mode,
	ePath:=PATH_GENERIC,
	bExecute:= ,
	tTimeout:=T#1s,
	hFile=> hFile);

fbFilePuts(
	sNetId:='',
	hFile:=hFile,
	sLine:= ,
	bExecute:= ,
	tTimeout:=t#1s);

fbFileClose(
	sNetId:='',
	hFile:=hFile,
	bExecute:= ,
	tTimeout:=t#1s);
END_FUNCTION_BLOCK

(* POU System/MPHandler/MPHandler, ST *)
PROGRAM MPHandler
VAR

	LocalFiles					: FB_EnumFindFileList;
	ExportFiles					: FB_EnumFindFileList;

	CreateDirectory			:FB_CreateDir;

	CopyFiles						:	FB_FileCopy;

	WriteXML						: FB_XmlSrvWriteByName;
	ReadXML							: FB_XmlSrvReadByName;


	LocalDirectory					: ARRAY[1..200] OF ST_FindFileEntry;
	ExportDirectory				: ARRAY[1..200] OF ST_FindFileEntry;

	i										:	DINT;
	j										:	DINT;

	FileNameSearchExport		:	STRING(255);
	FileNameSearchLocal		:	STRING(255);

	FileListUpdateExport		:	BOOL;
	FileListUpdateLocal		:	BOOL;

	BtnImport							:	VisuButton;
	BtnExport							:	VisuButton;


	StepExport					:	DINT;

	Delay : TON;

	NoOfTDFilesToCopy	:	DINT;
	AktFileToCopy			:	DINT;

	TempStringSource	:	STRING;
	TempStringTarget	:	STRING;

	Backslash						:	STRING :='\';

